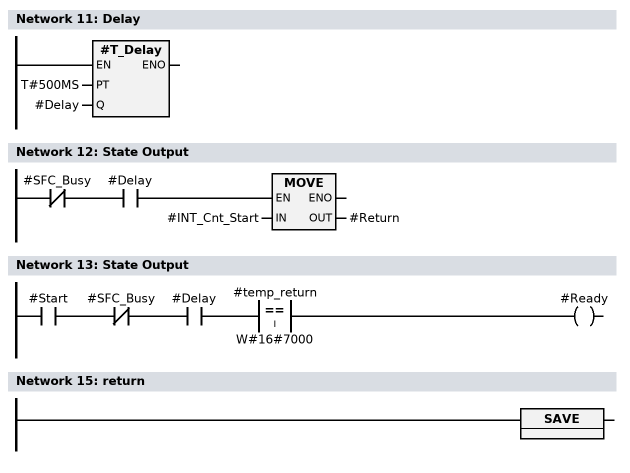
[picture p165: READ_DBL networks 11-15]
NETWORK
TITLE = Delay
      CALL  #T_Delay (
           PT                       := T#500MS,
           Q                        := #Delay);
      NOP   0;
NETWORK
TITLE = State Output
      AN    #SFC_Busy;
      A     #Delay;
      JNB   _007;
      L     #INT_Cnt_Start;
      T     #Return;
_007: NOP   0;
NETWORK
TITLE = State Output
      A     #Start;
      AN    #SFC_Busy;
      A     #Delay;
      A(;
      L     #temp_return;
      L     W#16#7000;
      ==I;
      );
      =     #Ready;
NETWORK
TITLE = restore register
      OPN   DB [#SysSave.DBNO];
      OPN   DI [#SysSave.DINO];
      LAR1  #SysSave.AR1;
      LAR2  #SysSave.AR2;
NETWORK
TITLE = return
      SET;
      SAVE;
END_FUNCTION_BLOCK

FUNCTION_BLOCK "WRITE_DBL"	// FB 193
TITLE = write to db on memory-card
//source-DB is on workarea of memory
//target-DB is on memory-card
VERSION : 0.1
VAR_INPUT
  DB_source : INT ;
  DB_target : INT ;
  Length : INT ;
  Start : BOOL ;
END_VAR
VAR_OUTPUT
  Return : INT ;
  Ready : BOOL ;
END_VAR
VAR
  imp_start : BOOL ;
  busy : BOOL ;
  puls_plus : BOOL ;
  puls_minus : BOOL ;
END_VAR
VAR_TEMP
  any_source : ANY ;
  any_target : ANY ;
  temp_rturn : INT ;
END_VAR
BEGIN
NETWORK
TITLE = create anypointer to source and target
//any to source
      L     W#16#1002;	//anytyp byte
      T     LW 0;
      L     #Length;	//number of bytes
      T     LW 2;
      L     #DB_source;	//number of DB-source 
      T     LW 4;
      L     0;	//begin in DB-source = byte 0
      SLD   3;
      OD    DW#16#84000000;	//constant
      T     LD 6;
//any to target
      L     W#16#1002;	//anytyp byte
      T     LW 10;
      L     #Length;	//number of bytes
      T     LW 12;
      L     #DB_target;	//number of DB-target
      T     LW 14;
      L     0;	//begin in DB-source = byte 0
      SLD   3;
      OD    DW#16#84000000;	//constant
      T     LD 16;
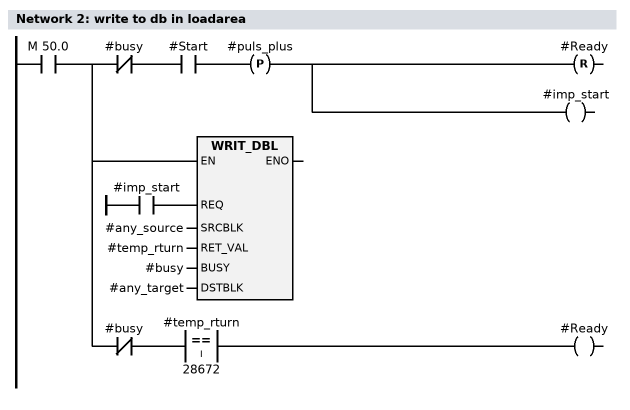
NETWORK
TITLE = write to db in loadarea
      A     M 50.0;
      =     L 22.0;
      A     L 22.0;
      AN    #busy;
      A(;
      A     #Start;
      BLD   100;
      FP    #puls_plus;
      );
      R     #Ready;
      =     #imp_start;
      A     #imp_start;
      =     L 22.1;
      BLD   103;
      A     L 22.0;
      JNB   _001;
      CALL  "WRIT_DBL" (
           REQ                      := L 22.1,
           SRCBLK                   := #any_source,
           RET_VAL                  := #temp_rturn,
           BUSY                     := #busy,
           DSTBLK                   := #any_target);
_001: NOP   0;
      A     L 22.0;
      AN    #busy;
      A(;
      L     #temp_rturn;
      L     28672;
      ==I;
      );
      =     #Ready;
END_FUNCTION_BLOCK

// FB 215: know-how protected block, not included

// FB 219: know-how protected block, not included

// FB 225: know-how protected block, not included

// FB 226: know-how protected block, not included

// FB 272: know-how protected block, not included

// FB 273: know-how protected block, not included

// FB 274: know-how protected block, not included

// FB 275: know-how protected block, not included

// FB 276: know-how protected block, not included

// FB 277: know-how protected block, not included

// FB 278: know-how protected block, not included

// FB 279: know-how protected block, not included

// FB 280: know-how protected block, not included

// FB 281: know-how protected block, not included

// FB 282: know-how protected block, not included

// FB 283: know-how protected block, not included

// FB 284: know-how protected block, not included

// FB 285: know-how protected block, not included

// FB 286: know-how protected block, not included

// FB 287: know-how protected block, not included

// FC 1: know-how protected block, not included

FUNCTION "Init" : VOID	// FC 2
TITLE = Program/PLC Init
VERSION : 0.1
VAR_TEMP
  ON : BOOL ;
  OFF : BOOL ;
END_VAR
BEGIN
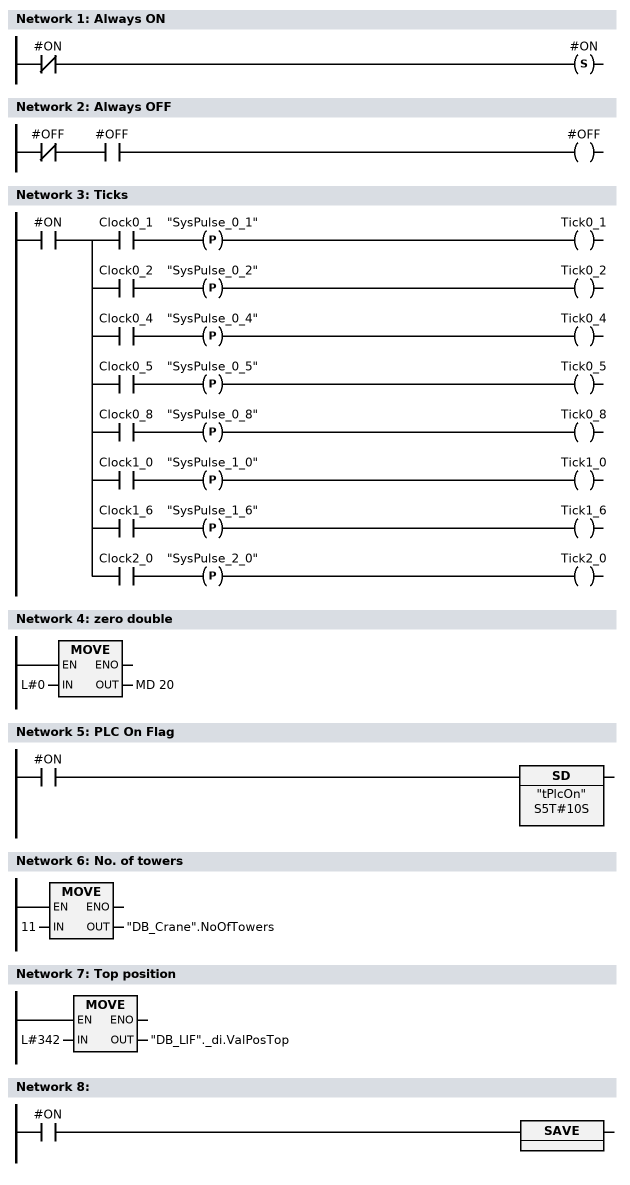
NETWORK
TITLE = Always ON
      AN    #ON;
      S     #ON;
NETWORK
TITLE = Always OFF
      AN    #OFF;
      A     #OFF;
      =     #OFF;
NETWORK
TITLE = Ticks
      A     #ON;
      =     L 1.0;
      A     L 1.0;
      A     "Clock0_1";
      FP    "SysPulse_0_1";
      =     "Tick0_1";
      A     L 1.0;
      A     "Clock0_2";
      FP    "SysPulse_0_2";
      =     "Tick0_2";
      A     L 1.0;
      A     "Clock0_4";
      FP    "SysPulse_0_4";
      =     "Tick0_4";
      A     L 1.0;
      A     "Clock0_5";
      FP    "SysPulse_0_5";
      =     "Tick0_5";
      A     L 1.0;
      A     "Clock0_8";
      FP    "SysPulse_0_8";
      =     "Tick0_8";
      A     L 1.0;
      A     "Clock1_0";
      FP    "SysPulse_1_0";
      =     "Tick1_0";
      A     L 1.0;
      A     "Clock1_6";
      FP    "SysPulse_1_6";
      =     "Tick1_6";
      A     L 1.0;
      A     "Clock2_0";
      FP    "SysPulse_2_0";
      =     "Tick2_0";
NETWORK
TITLE = zero double
      L     L#0;
      T     MD 20;
      NOP   0;
NETWORK
TITLE = PLC On Flag
      A     #ON;
      L     S5T#10S;
      SD    "tPlcOn";
NETWORK
TITLE = No. of towers
      L     11;
      T     "DB_Crane".NoOfTowers;
      NOP   0;
NETWORK
TITLE = Top position
      L     L#342;
      T     "DB_LIF"._di.ValPosTop;
      NOP   0;
NETWORK
TITLE =
      A     #ON;
      SAVE;
END_FUNCTION

// FC 5: know-how protected block, not included

// FC 6: know-how protected block, not included

// FC 8: know-how protected block, not included

FUNCTION "OpHours" : VOID	// FC 9
VERSION : 0.1
VAR_INPUT
  IN_xMoving : BOOL ;
  IN_xTick_1sec : BOOL ;
  IN_xResetServHours : BOOL ;
  IN_diServHoursPrest : DINT ;
END_VAR
VAR_IN_OUT
  INOUT_iWorkSec : INT ;
  INOUT_iServSec : INT ;
  INOUT_diWorkHours : DINT ;
  INOUT_diServHours : DINT ;
END_VAR
BEGIN
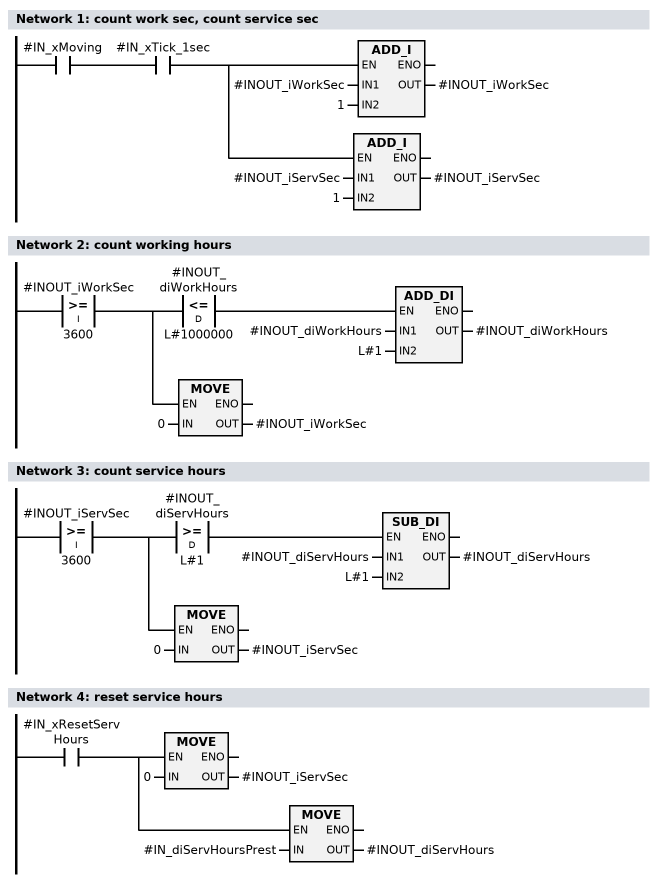
NETWORK
TITLE = count work sec, count service sec
      A     #IN_xMoving;
      A     #IN_xTick_1sec;
      =     L 0.0;
      A     L 0.0;
      JNB   _001;
      L     #INOUT_iWorkSec;
      L     1;
      +I;
      T     #INOUT_iWorkSec;
_001: NOP   0;
      A     L 0.0;
      JNB   _002;
      L     #INOUT_iServSec;
      L     1;
      +I;
      T     #INOUT_iServSec;
_002: NOP   0;
NETWORK
TITLE = count working hours
      L     #INOUT_iWorkSec;
      L     3600;
      >=I;
      =     L 0.0;
      A     L 0.0;
      A(;
      L     #INOUT_diWorkHours;
      L     L#1000000;
      <=D;
      );
      JNB   _003;
      L     #INOUT_diWorkHours;
      L     L#1;
      +D;
      T     #INOUT_diWorkHours;
_003: NOP   0;
      A     L 0.0;
      JNB   _004;
      L     0;
      T     #INOUT_iWorkSec;
_004: NOP   0;
NETWORK
TITLE = count service hours
      L     #INOUT_iServSec;
      L     3600;
      >=I;
      =     L 0.0;
      A     L 0.0;
      A(;
      L     #INOUT_diServHours;
      L     L#1;
      >=D;
      );
      JNB   _005;
      L     #INOUT_diServHours;
      L     L#1;
      -D;
      T     #INOUT_diServHours;
_005: NOP   0;
      A     L 0.0;
      JNB   _006;
      L     0;
      T     #INOUT_iServSec;
_006: NOP   0;
NETWORK
TITLE = reset service hours
      A     #IN_xResetServHours;
      =     L 0.0;
      A     L 0.0;
      JNB   _007;
      L     0;
      T     #INOUT_iServSec;
_007: NOP   0;
      A     L 0.0;
      JNB   _008;
      L     #IN_diServHoursPrest;
      T     #INOUT_diServHours;
_008: NOP   0;
END_FUNCTION

// FC 10: know-how protected block, not included

FUNCTION "AbsEncoder" : VOID	// FC 11
TITLE = AbsEncoder
//calculate position value depend from encoder resolution
VERSION : 0.1
VAR_INPUT
  IN_DW_ProcessData : DWORD ;
  IN_DINT_Turn100 : DINT ;
  IN_DINT_PresetVal : DINT ;
  IN_Resolution_4096 : BOOL ;
  IN_Resolution_8192 : BOOL ;
  IN_BOOL_Preset : BOOL ;
END_VAR
VAR_OUTPUT
  OUT_DINT_EncMm : DINT ;
  OUT_DW_ProcessData : DWORD ;
END_VAR
VAR_TEMP
  TEMP_DINT_WayByFullTurns : DINT ;
  TEMP_DINT_WayByActTurn : DINT ;
  TEMP_DINT_Resolution : DINT ;
  TEMP_DW_01 : DWORD ;
  TEMP_DW_00 : DWORD ;
  TEMP_DW_Mask1 : DWORD ;
  TEMP_W_Mask2 : WORD ;
  TEMP_DW_Mask3 : DWORD ;
  TEMP_DINT_00 : DINT ;
  TEMP_DINT_PresetTurns : DINT ;
  TEMP_DINT_PresetVal100 : DINT ;
  TEMP_DINT_PresetAngle : DINT ;
  ON : BOOL ;
  TEMP_BOOL_RetValFault : BOOL ;
END_VAR
BEGIN
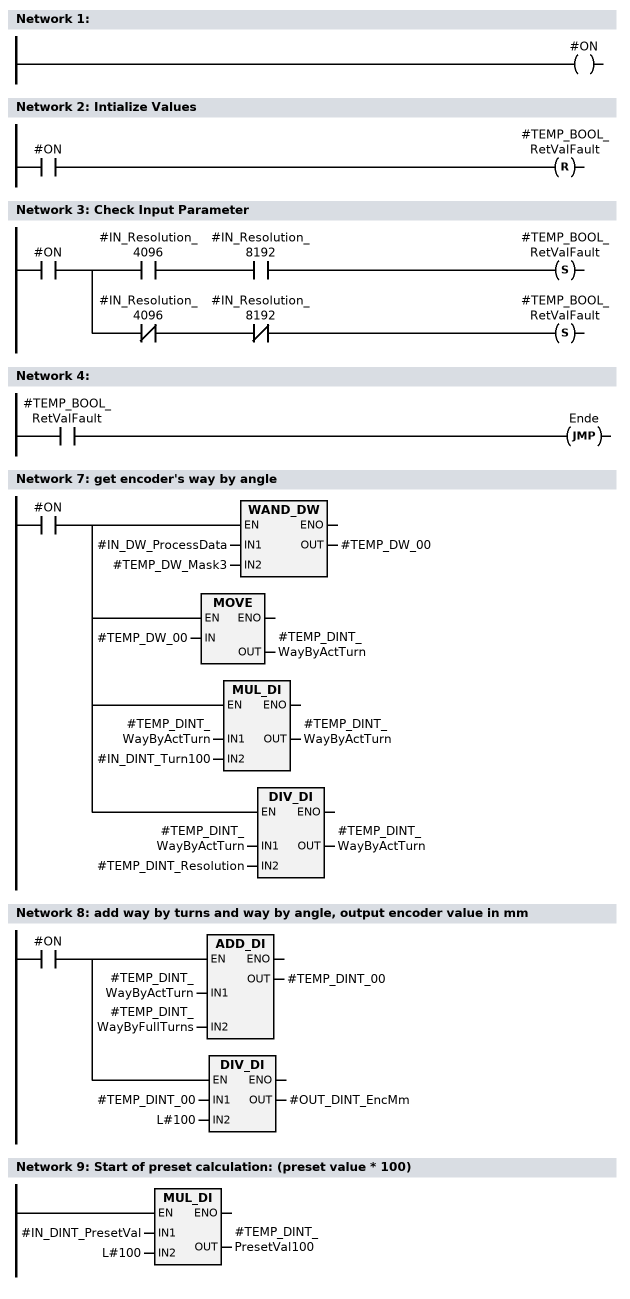
NETWORK
TITLE =
      SET;
      =     #ON;
NETWORK
TITLE = Intialize Values
      A     #ON;
      R     #TEMP_BOOL_RetValFault;
NETWORK
TITLE = Check Input Parameter
      A     #ON;
      =     L 47.0;
      A     L 47.0;
      A     #IN_Resolution_4096;
      A     #IN_Resolution_8192;
      S     #TEMP_BOOL_RetValFault;
      A     L 47.0;
      AN    #IN_Resolution_4096;
      AN    #IN_Resolution_8192;
      S     #TEMP_BOOL_RetValFault;
NETWORK
TITLE =
      A     #TEMP_BOOL_RetValFault;
      JC    Ende;
NETWORK
TITLE =
      A     #ON;
      =     L 47.0;
      A     L 47.0;
      A     #IN_Resolution_4096;
      =     L 47.1;
      A(;
      A(;
      A     L 47.1;
      JNB   _001;
      L     DW#16#1FFF000;
      T     #TEMP_DW_Mask1;
      SET;
      SAVE;
      CLR;
_001: A     BR;
      );
      JNB   _002;
      L     W#16#C;
      T     #TEMP_W_Mask2;
      SET;
      SAVE;
      CLR;
_002: A     BR;
      );
      JNB   _003;
      L     DW#16#FFF;
      T     #TEMP_DW_Mask3;
_003: NOP   0;
      A     L 47.1;
      JNB   _004;
      L     L#4096;
      T     #TEMP_DINT_Resolution;
_004: NOP   0;
      A     L 47.0;
      A     #IN_Resolution_8192;
      =     L 47.1;
      A(;
      A(;
      A     L 47.1;
      JNB   _005;
      L     DW#16#1FFE000;
      T     #TEMP_DW_Mask1;
      SET;
      SAVE;
      CLR;
_005: A     BR;
      );
      JNB   _006;
      L     W#16#D;
      T     #TEMP_W_Mask2;
      SET;
      SAVE;
      CLR;
_006: A     BR;
      );
      JNB   _007;
      L     DW#16#1FFF;
      T     #TEMP_DW_Mask3;
_007: NOP   0;
      A     L 47.1;
      JNB   _008;
      L     L#8192;
      T     #TEMP_DINT_Resolution;
_008: NOP   0;
NETWORK
TITLE = Start of actual mm-calculation: get encoder's way by full turns
      A     #ON;
      =     L 47.0;
      A     L 47.0;
      JNB   _009;
      L     #IN_DW_ProcessData;
      L     #TEMP_DW_Mask1;
      AD;
      T     #TEMP_DW_00;
_009: NOP   0;
      A     L 47.0;
      JNB   _00a;
      L     #TEMP_W_Mask2;
      L     #TEMP_DW_00;
      SRD;
      T     #TEMP_DW_00;
_00a: NOP   0;
      A     L 47.0;
      JNB   _00b;
      L     #TEMP_DW_00;
      T     #TEMP_DINT_WayByFullTurns;
_00b: NOP   0;
      A     L 47.0;
      JNB   _00c;
      L     #TEMP_DINT_WayByFullTurns;
      L     #IN_DINT_Turn100;
      *D;
      T     #TEMP_DINT_WayByFullTurns;
_00c: NOP   0;
NETWORK
TITLE = get encoder's way by angle
      A     #ON;
      =     L 47.0;
      A     L 47.0;
      JNB   _00d;
      L     #IN_DW_ProcessData;
      L     #TEMP_DW_Mask3;
      AD;
      T     #TEMP_DW_00;
_00d: NOP   0;
      A     L 47.0;
      JNB   _00e;
      L     #TEMP_DW_00;
      T     #TEMP_DINT_WayByActTurn;
_00e: NOP   0;
      A     L 47.0;
      JNB   _00f;
      L     #TEMP_DINT_WayByActTurn;
      L     #IN_DINT_Turn100;
      *D;
      T     #TEMP_DINT_WayByActTurn;
_00f: NOP   0;
      A     L 47.0;
      JNB   _010;
      L     #TEMP_DINT_WayByActTurn;
      L     #TEMP_DINT_Resolution;
      /D;
      T     #TEMP_DINT_WayByActTurn;
_010: NOP   0;
NETWORK
TITLE = add way by turns and way by angle, output encoder value in mm
      A     #ON;
      =     L 47.0;
      A     L 47.0;
      JNB   _011;
      L     #TEMP_DINT_WayByActTurn;
      L     #TEMP_DINT_WayByFullTurns;
      +D;
      T     #TEMP_DINT_00;
_011: NOP   0;
      A     L 47.0;
      JNB   _012;
      L     #TEMP_DINT_00;
      L     L#100;
      /D;
      T     #OUT_DINT_EncMm;
_012: NOP   0;
NETWORK
TITLE = Start of preset calculation: (preset value * 100)
      L     #IN_DINT_PresetVal;
      L     L#100;
      *D;
      T     #TEMP_DINT_PresetVal100;
      NOP   0;
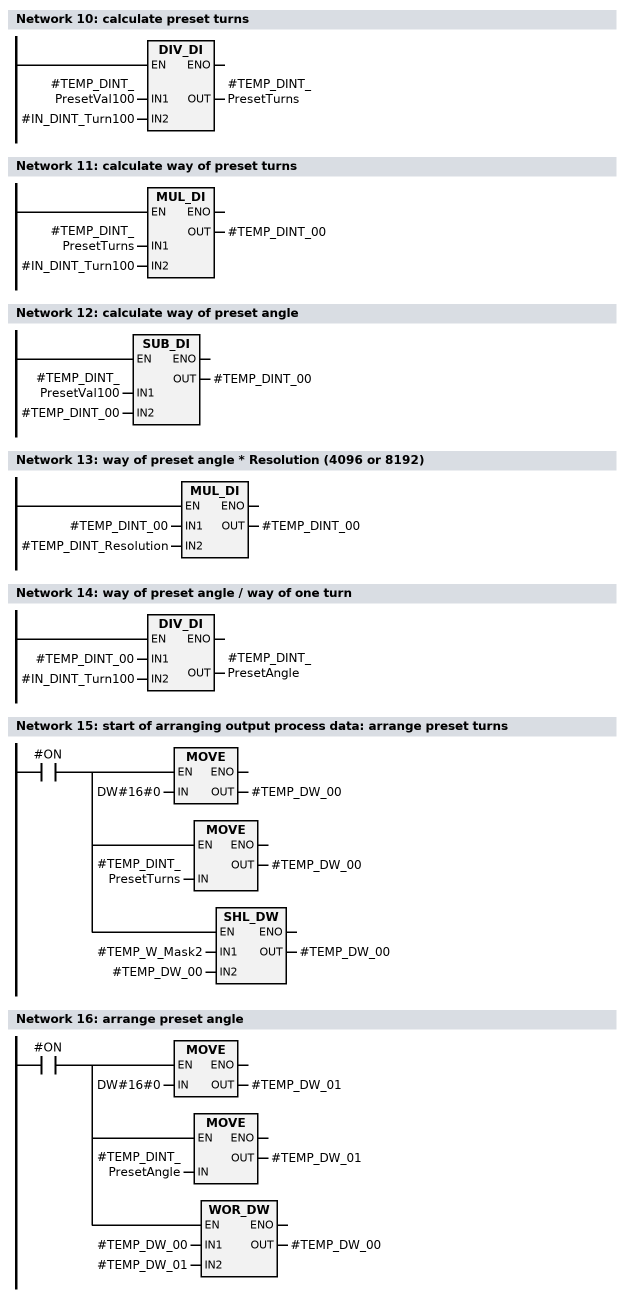
NETWORK
TITLE = calculate preset turns
      L     #TEMP_DINT_PresetVal100;
      L     #IN_DINT_Turn100;
      /D;
      T     #TEMP_DINT_PresetTurns;
      NOP   0;
NETWORK
TITLE = calculate way of preset turns
      L     #TEMP_DINT_PresetTurns;
      L     #IN_DINT_Turn100;
      *D;
      T     #TEMP_DINT_00;
      NOP   0;
NETWORK
TITLE = calculate way of preset angle 
      L     #TEMP_DINT_PresetVal100;
      L     #TEMP_DINT_00;
      -D;
      T     #TEMP_DINT_00;
      NOP   0;
NETWORK
TITLE = way of preset angle * Resolution (4096 or 8192)
      L     #TEMP_DINT_00;
      L     #TEMP_DINT_Resolution;
      *D;
      T     #TEMP_DINT_00;
      NOP   0;
NETWORK
TITLE = way of preset angle / way of one turn
      L     #TEMP_DINT_00;
      L     #IN_DINT_Turn100;
      /D;
      T     #TEMP_DINT_PresetAngle;
      NOP   0;
NETWORK
TITLE = start of arranging output process data: arrange preset turns
      A     #ON;
      =     L 47.0;
      A     L 47.0;
      JNB   _013;
      L     DW#16#0;
      T     #TEMP_DW_00;
_013: NOP   0;
      A     L 47.0;
      JNB   _014;
      L     #TEMP_DINT_PresetTurns;
      T     #TEMP_DW_00;
_014: NOP   0;
      A     L 47.0;
      JNB   _015;
      L     #TEMP_W_Mask2;
      L     #TEMP_DW_00;
      SLD;
      T     #TEMP_DW_00;
_015: NOP   0;
NETWORK
TITLE = arrange preset angle
      A     #ON;
      =     L 47.0;
      A     L 47.0;
      JNB   _016;
      L     DW#16#0;
      T     #TEMP_DW_01;
_016: NOP   0;
      A     L 47.0;
      JNB   _017;
      L     #TEMP_DINT_PresetAngle;
      T     #TEMP_DW_01;
_017: NOP   0;
      A     L 47.0;
      JNB   _018;
      L     #TEMP_DW_00;
      L     #TEMP_DW_01;
      OD;
      T     #TEMP_DW_00;
_018: NOP   0;
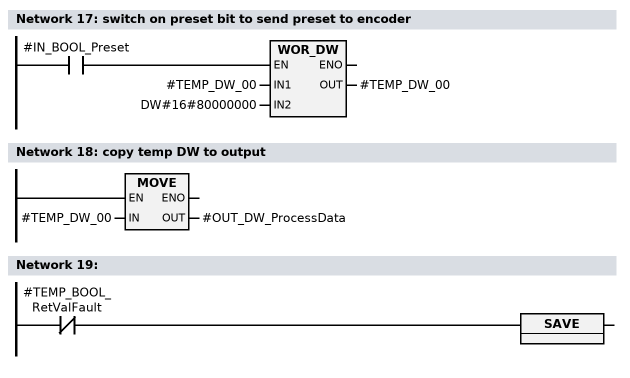
NETWORK
TITLE = switch on preset bit to send preset to encoder
      A     #IN_BOOL_Preset;
      JNB   _019;
      L     #TEMP_DW_00;
      L     DW#16#80000000;
      OD;
      T     #TEMP_DW_00;
_019: NOP   0;
NETWORK
TITLE = copy temp DW to output 
      L     #TEMP_DW_00;
      T     #OUT_DW_ProcessData;
      NOP   0;
NETWORK
TITLE =
Ende: AN    #TEMP_BOOL_RetValFault;
      SAVE;
END_FUNCTION

FUNCTION "Motor_2_frequ" : VOID	// FC 12
VERSION : 0.1
VAR_INPUT
  IN_x_Release : BOOL ;
  IN_BOOL_ServLeft : BOOL ;
  IN_BOOL_ServRight : BOOL ;
  IN_BOOL_ServMode : BOOL ;
  IN_StartPosMode : BOOL ;
  IN_TargetVal : DINT ;
  IN_ActPos : DINT ;
  IN_SlowWin : DINT ;
  IN_StopWin : DINT ;
  IN_PosWin : DINT ;
END_VAR
VAR_OUTPUT
  OUT_BOOL_FastFrequ : BOOL ;
  OUT_BOOL_Pos_OK : BOOL ;
END_VAR
VAR_IN_OUT
  INOUT_x_Minus : BOOL ;
  INOUT_x_Plus : BOOL ;
END_VAR
VAR_TEMP
  TEMP_DINT_00 : DINT ;
  TMP_x_InPosition : BOOL ;
  TMP_x_Slow : BOOL ;
  TMP_x_PosOk : BOOL ;
END_VAR
BEGIN
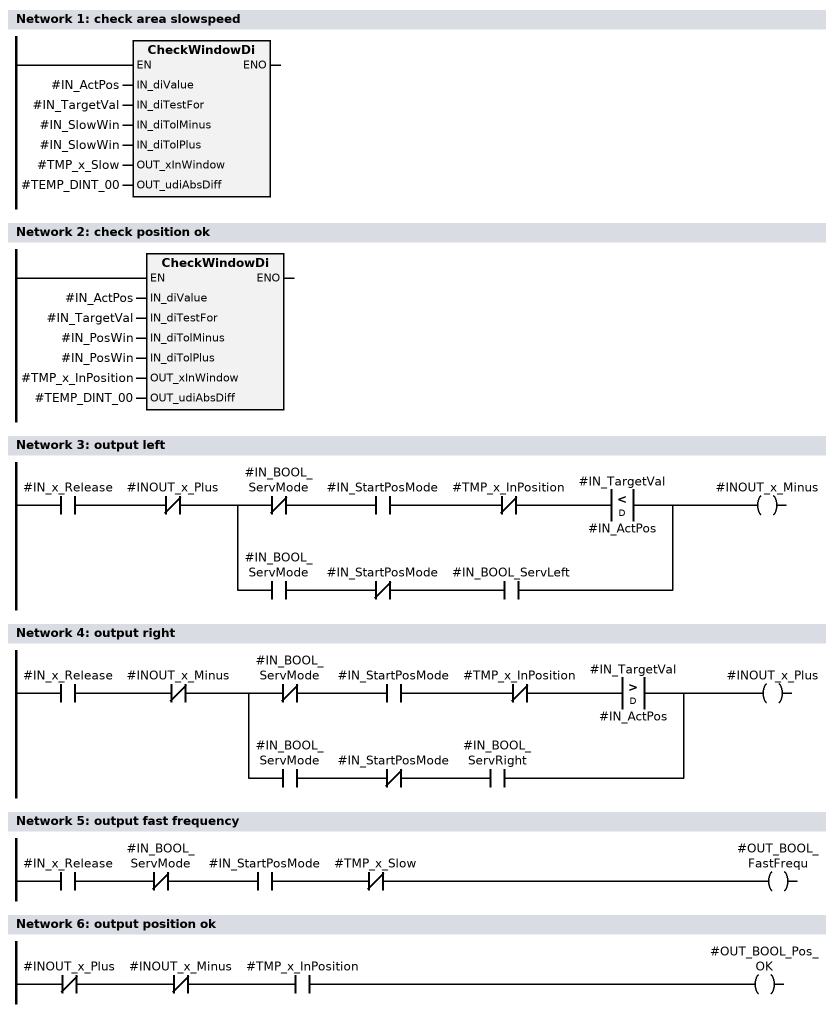
NETWORK
TITLE = check area slowspeed
      CALL  "CheckWindowDi" (
           IN_diValue               := #IN_ActPos,
           IN_diTestFor             := #IN_TargetVal,
           IN_diTolMinus            := #IN_SlowWin,
           IN_diTolPlus             := #IN_SlowWin,
           OUT_xInWindow            := #TMP_x_Slow,
           OUT_udiAbsDiff           := #TEMP_DINT_00);
      NOP   0;
NETWORK
TITLE = check position ok
      CALL  "CheckWindowDi" (
           IN_diValue               := #IN_ActPos,
           IN_diTestFor             := #IN_TargetVal,
           IN_diTolMinus            := #IN_PosWin,
           IN_diTolPlus             := #IN_PosWin,
           OUT_xInWindow            := #TMP_x_InPosition,
           OUT_udiAbsDiff           := #TEMP_DINT_00);
      NOP   0;
NETWORK
TITLE = output left
      A     #IN_x_Release;
      AN    #INOUT_x_Plus;
      A(;
      AN    #IN_BOOL_ServMode;
      A     #IN_StartPosMode;
      AN    #TMP_x_InPosition;
      A(;
      L     #IN_TargetVal;
      L     #IN_ActPos;
      <D;
      );
      O;
      A     #IN_BOOL_ServMode;
      AN    #IN_StartPosMode;
      A     #IN_BOOL_ServLeft;
      );
      =     #INOUT_x_Minus;
NETWORK
TITLE = output right
      A     #IN_x_Release;
      AN    #INOUT_x_Minus;
      A(;
      AN    #IN_BOOL_ServMode;
      A     #IN_StartPosMode;
      AN    #TMP_x_InPosition;
      A(;
      L     #IN_TargetVal;
      L     #IN_ActPos;
      >D;
      );
      O;
      A     #IN_BOOL_ServMode;
      AN    #IN_StartPosMode;
      A     #IN_BOOL_ServRight;
      );
      =     #INOUT_x_Plus;
NETWORK
TITLE = output fast frequency 
      A     #IN_x_Release;
      AN    #IN_BOOL_ServMode;
      A     #IN_StartPosMode;
      AN    #TMP_x_Slow;
      =     #OUT_BOOL_FastFrequ;
NETWORK
TITLE = output position ok
      AN    #INOUT_x_Plus;
      AN    #INOUT_x_Minus;
      A     #TMP_x_InPosition;
      =     #OUT_BOOL_Pos_OK;
END_FUNCTION

// FC 15: know-how protected block, not included

FUNCTION "Scan_BRI" : VOID	// FC 21
TITLE = scan positions bridge
VERSION : 0.1
VAR_INPUT
  in_i_DBNo : INT ;
  in_i_ActRow : INT ;
  in_i_NoOfDataSets : INT ;
  in_di_DatSetLenght : DINT ;
  in_di_ActAxisPos : DINT ;
  in_di_DataStartByte : DINT ;
  in_di_AreaWin : DINT ;
  in_di_PosWin : DINT ;
END_VAR
VAR_OUTPUT
  out_i_SetNo : INT ;
  out_i_AreaNo : INT ;
  out_b_InArea : BOOL ;
  out_b_InPos : BOOL ;
  out_i_LIF_DBNo : INT ;
  out_i_LIF_DBNo_2 : INT ;
END_VAR
VAR_TEMP
  Save_AR1 : DWORD ;
  Save_AR2 : DWORD ;
  tmp_di_1 : DINT ;
  tmp_di_2 : DINT ;
  tmp_di_Pointer : DINT ;
  tmp_di_PosVal : DINT ;
  tmp_i_PosNo : INT ;
  tmp_i_PosNoVal : INT ;
  tmp_i_DBNo : INT ;
  tmp_i_1 : INT ;
  tmp_i_LIF_DBNo : INT ;
  tmp_i_LIF_DBNo_2 : INT ;
  tmp_i_offsetPointer : INT ;
  ON : BOOL ;
  OFF : BOOL ;
  tmp_b_LoopBrake : BOOL ;
  err_input : BOOL ;
END_VAR
BEGIN
NETWORK
TITLE = save register
      TAR1  #Save_AR1;
      TAR2  #Save_AR2;
NETWORK
TITLE = on/off
      SET;
      =     #ON;
      CLR;
      =     #OFF;
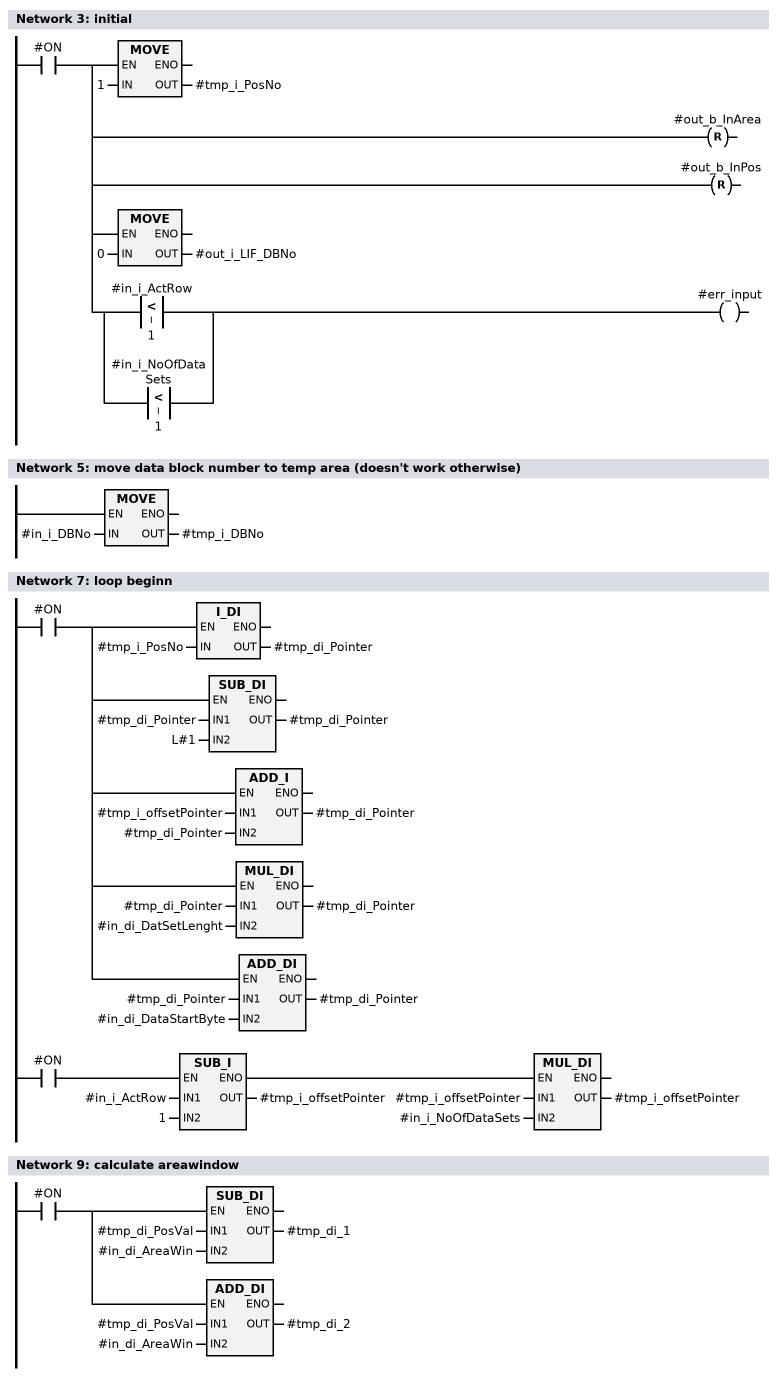
NETWORK
TITLE = initial
//set loopcounter to 0
//reset outputs
      A     #ON;
      =     L 40.0;
      A     L 40.0;
      JNB   _001;
      L     1;
      T     #tmp_i_PosNo;
_001: NOP   0;
      A     L 40.0;
      BLD   102;
      R     #out_b_InArea;
      A     L 40.0;
      BLD   102;
      R     #out_b_InPos;
      A     L 40.0;
      JNB   _002;
      L     0;
      T     #out_i_LIF_DBNo;
_002: NOP   0;
      A     L 40.0;
      A(;
      O(;
      L     #in_i_ActRow;
      L     1;
      <I;
      );
      O(;
      L     #in_i_NoOfDataSets;
      L     1;
      <I;
      );
      );
      =     #err_input;
NETWORK
TITLE =
      AN    #err_input;
      JC    NoEr;	// On Error CLR all Outputs
      L     0;
      T     #out_i_SetNo;
      T     #out_i_AreaNo;
      T     #out_i_LIF_DBNo;
      T     #out_i_LIF_DBNo_2;
      A     #OFF;
      =     #out_b_InArea;
      =     #out_b_InPos;
      BEU;
NoEr: NOP   0;
NETWORK
TITLE = move data block number to temp area (doesn't work otherwise)
//doesn't work otherwise
      L     #in_i_DBNo;
      T     #tmp_i_DBNo;
      NOP   0;
NETWORK
TITLE = open DB
      OPN   DB [#tmp_i_DBNo];
NETWORK
TITLE = loop beginn
//calculate pointer to positionvalue
//insert calculating rows [2016 TH]
scbr: A     #ON;
      =     L 39.0;
      A     L 39.0;
      JNB   _003;
      L     #tmp_i_PosNo;
      ITD;
      T     #tmp_di_Pointer;
_003: NOP   0;
      A     L 39.0;
      JNB   _004;
      L     #tmp_di_Pointer;
      L     L#1;
      -D;
      T     #tmp_di_Pointer;
_004: NOP   0;
      A(;
      A     L 39.0;
      JNB   _005;
      L     #in_i_ActRow;
      L     1;
      -I;
      T     #tmp_i_offsetPointer;
      AN    OV;
      SAVE;
      CLR;
_005: A     BR;
      );
      JNB   _006;
      L     #tmp_i_offsetPointer;
      L     #in_i_NoOfDataSets;
      *D;
      T     #tmp_i_offsetPointer;
_006: NOP   0;
      A     L 39.0;
      JNB   _007;
      L     #tmp_i_offsetPointer;
      L     #tmp_di_Pointer;
      +I;
      T     #tmp_di_Pointer;
_007: NOP   0;
      A     L 39.0;
      JNB   _008;
      L     #tmp_di_Pointer;
      L     #in_di_DatSetLenght;
      *D;
      T     #tmp_di_Pointer;
_008: NOP   0;
      A     L 39.0;
      JNB   _009;
      L     #tmp_di_Pointer;
      L     #in_di_DataStartByte;
      +D;
      T     #tmp_di_Pointer;
_009: NOP   0;
NETWORK
TITLE = get positionvalue 
      L     #tmp_di_Pointer;	// load pointer
      SLD   3;	// shift left 3 bits to achieve pointer format
      LAR1;	// load adressregister 1 with pointer
      L     DBD [AR1,P#2.0];	// load position from DataBlock
      T     #tmp_di_PosVal;	// Transfer to temp for window check
      L     DBW [AR1,P#0.0];
      T     #tmp_i_PosNoVal;
      L     DBW [AR1,P#6.0];	// LIF DB number
      T     #tmp_i_LIF_DBNo;
      L     DBW [AR1,P#8.0];	// LIF DB number
      T     #tmp_i_LIF_DBNo_2;
NETWORK
TITLE = calculate areawindow
      A     #ON;
      =     L 40.0;
      A     L 40.0;
      JNB   _00a;
      L     #tmp_di_PosVal;
      L     #in_di_AreaWin;
      -D;
      T     #tmp_di_1;
_00a: NOP   0;
      A     L 40.0;
      JNB   _00b;
      L     #tmp_di_PosVal;
      L     #in_di_AreaWin;
      +D;
      T     #tmp_di_2;
_00b: NOP   0;
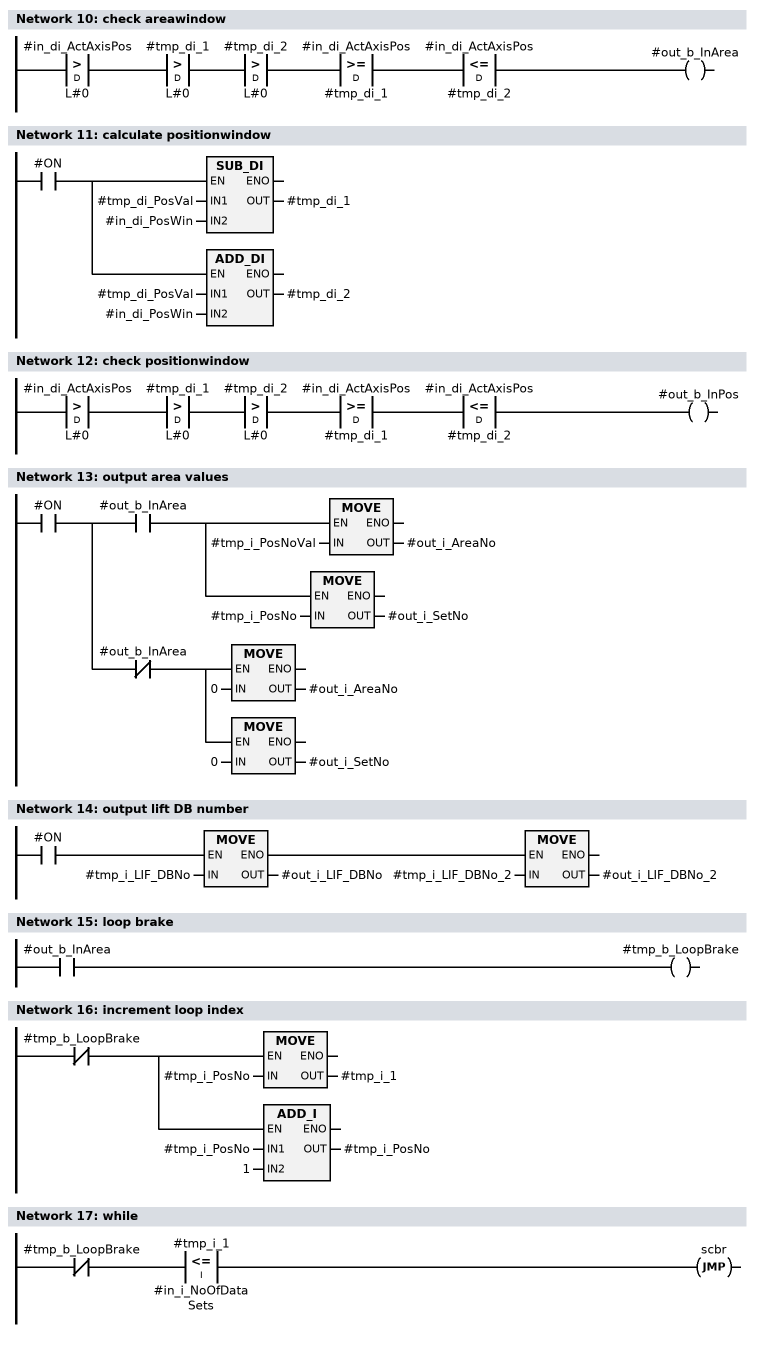
NETWORK
TITLE = check areawindow
      A(;
      L     #in_di_ActAxisPos;
      L     L#0;
      >D;
      );
      A(;
      L     #tmp_di_1;
      L     L#0;
      >D;
      );
      A(;
      L     #tmp_di_2;
      L     L#0;
      >D;
      );
      A(;
      L     #in_di_ActAxisPos;
      L     #tmp_di_1;
      >=D;
      );
      A(;
      L     #in_di_ActAxisPos;
      L     #tmp_di_2;
      <=D;
      );
      =     #out_b_InArea;
NETWORK
TITLE = calculate positionwindow
      A     #ON;
      =     L 40.0;
      A     L 40.0;
      JNB   _00c;
      L     #tmp_di_PosVal;
      L     #in_di_PosWin;
      -D;
      T     #tmp_di_1;
_00c: NOP   0;
      A     L 40.0;
      JNB   _00d;
      L     #tmp_di_PosVal;
      L     #in_di_PosWin;
      +D;
      T     #tmp_di_2;
_00d: NOP   0;
NETWORK
TITLE = check positionwindow
      A(;
      L     #in_di_ActAxisPos;
      L     L#0;
      >D;
      );
      A(;
      L     #tmp_di_1;
      L     L#0;
      >D;
      );
      A(;
      L     #tmp_di_2;
      L     L#0;
      >D;
      );
      A(;
      L     #in_di_ActAxisPos;
      L     #tmp_di_1;
      >=D;
      );
      A(;
      L     #in_di_ActAxisPos;
      L     #tmp_di_2;
      <=D;
      );
      =     #out_b_InPos;
NETWORK
TITLE = output area values
      A     #ON;
      =     L 40.0;
      A     L 40.0;
      A     #out_b_InArea;
      =     L 40.1;
      A     L 40.1;
      JNB   _00e;
      L     #tmp_i_PosNoVal;
      T     #out_i_AreaNo;
_00e: NOP   0;
      A     L 40.1;
      JNB   _00f;
      L     #tmp_i_PosNo;
      T     #out_i_SetNo;
_00f: NOP   0;
      A     L 40.0;
      AN    #out_b_InArea;
      =     L 40.1;
      A     L 40.1;
      JNB   _010;
      L     0;
      T     #out_i_AreaNo;
_010: NOP   0;
      A     L 40.1;
      JNB   _011;
      L     0;
      T     #out_i_SetNo;
_011: NOP   0;
NETWORK
TITLE = output lift DB number
      A(;
      A     #ON;
      JNB   _012;
      L     #tmp_i_LIF_DBNo;
      T     #out_i_LIF_DBNo;
      SET;
      SAVE;
      CLR;
_012: A     BR;
      );
      JNB   _013;
      L     #tmp_i_LIF_DBNo_2;
      T     #out_i_LIF_DBNo_2;
_013: NOP   0;
NETWORK
TITLE = loop brake
      A     #out_b_InArea;
      =     #tmp_b_LoopBrake;
NETWORK
TITLE = increment loop index
      AN    #tmp_b_LoopBrake;
      =     L 40.0;
      A     L 40.0;
      JNB   _014;
      L     #tmp_i_PosNo;
      T     #tmp_i_1;
_014: NOP   0;
      A     L 40.0;
      JNB   _015;
      L     #tmp_i_PosNo;
      L     1;
      +I;
      T     #tmp_i_PosNo;
_015: NOP   0;
NETWORK
TITLE = while 
      AN    #tmp_b_LoopBrake;
      A(;
      L     #tmp_i_1;
      L     #in_i_NoOfDataSets;
      <=I;
      );
      JC    scbr;
NETWORK
TITLE = restore register
      LAR1  #Save_AR1;
      LAR2  #Save_AR2;
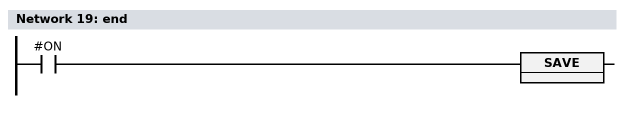
NETWORK
TITLE = end
      A     #ON;
      SAVE;
END_FUNCTION

FUNCTION "Scan_BRI_MAN" : VOID	// FC 22
TITLE = scan positions bridge
VERSION : 1.0
VAR_INPUT
  in_i_DBNo : INT ;
  in_i_ActRow : INT ;
  in_i_NoOfDataSets : INT ;
  in_di_DatSetLenght : DINT ;
  in_di_DataStartByte : DINT ;
  in_di_ActAxisPos : DINT ;
END_VAR
VAR_OUTPUT
  out_di_PrevPos : DINT ;
  out_di_ActPos : DINT ;
  out_di_NextPos : DINT ;
  out_di_MinPos : DINT ;
  out_di_MaxPos : DINT ;
  out_i_PrevPosNo : INT ;
  out_i_NextPosNo : INT ;
  out_i_MinPosNo : INT ;
  out_i_MaxPosNo : INT ;
END_VAR
VAR_TEMP
  Save_AR1 : DWORD ;
  Save_AR2 : DWORD ;
  tmp_di_1 : DINT ;
  tmp_di_Pointer : DINT ;
  tmp_di_PosVal : DINT ;
  tmp_di_PosData : DINT ;
  tmp_di_PosDataPlus : DINT ;
  tmp_di_PosDataMinus : DINT ;
  tmp_di_PosDataLow : DINT ;
  tmp_di_PosDataHigh : DINT ;
  tmp_di_PrevPos : DINT ;
  tmp_di_NextPos : DINT ;
  tmp_i_Counter : INT ;
  tmp_i_DBNo : INT ;
  tmp_i_PosNo : INT ;
  tmp_i_PosDataNo : INT ;
  tmp_i_PrevPosNo : INT ;
  tmp_i_NextPosNo : INT ;
  tmp_i_MinPosNo : INT ;
  tmp_i_MaxPosNo : INT ;
  tmp_i_1 : INT ;
  tmp_i_offsetPointer : INT ;
  TEMP1 : BOOL ;
  ON : BOOL ;
  OFF : BOOL ;
  err_input : BOOL ;
END_VAR
BEGIN
NETWORK
TITLE = save register
      TAR1  #Save_AR1;
      TAR2  #Save_AR2;
NETWORK
TITLE = on/off
      SET;
      =     #ON;
      CLR;
      =     #OFF;
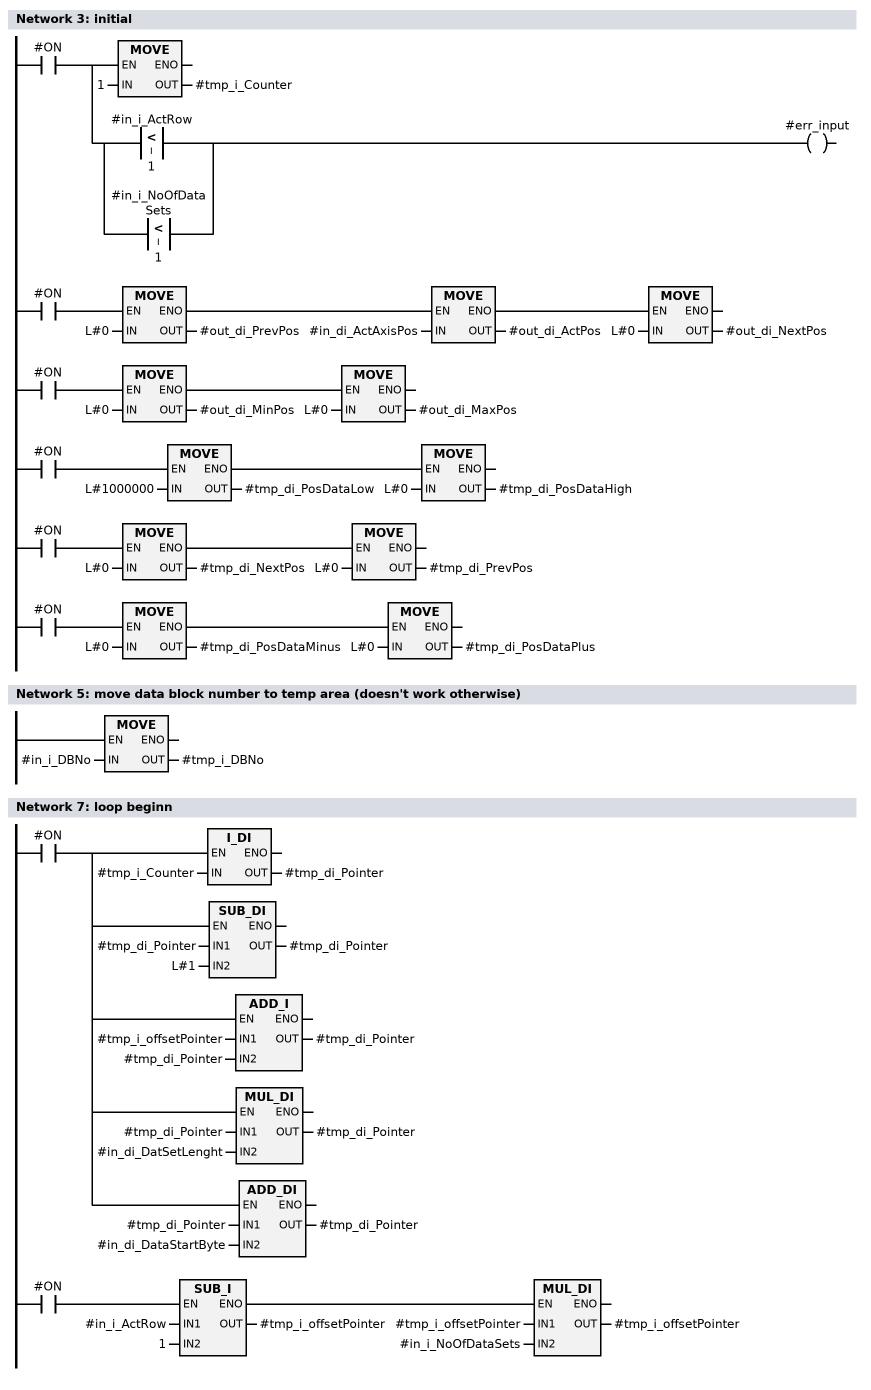
NETWORK
TITLE = initial
//set loopcounter to 0
//reset outputs
      A     #ON;
      =     L 70.0;
      A     L 70.0;
      JNB   _001;
      L     1;
      T     #tmp_i_Counter;
_001: NOP   0;
      A(;
      A(;
      A     L 70.0;
      JNB   _002;
      L     L#0;
      T     #out_di_PrevPos;
      SET;
      SAVE;
      CLR;
_002: A     BR;
      );
      JNB   _003;
      L     #in_di_ActAxisPos;
      T     #out_di_ActPos;
      SET;
      SAVE;
      CLR;
_003: A     BR;
      );
      JNB   _004;
      L     L#0;
      T     #out_di_NextPos;
_004: NOP   0;
      A(;
      A     L 70.0;
      JNB   _005;
      L     L#0;
      T     #out_di_MinPos;
      SET;
      SAVE;
      CLR;
_005: A     BR;
      );
      JNB   _006;
      L     L#0;
      T     #out_di_MaxPos;
_006: NOP   0;
      A(;
      A     L 70.0;
      JNB   _007;
      L     L#1000000;
      T     #tmp_di_PosDataLow;
      SET;
      SAVE;
      CLR;
_007: A     BR;
      );
      JNB   _008;
      L     L#0;
      T     #tmp_di_PosDataHigh;
_008: NOP   0;
      A(;
      A     L 70.0;
      JNB   _009;
      L     L#0;
      T     #tmp_di_NextPos;
      SET;
      SAVE;
      CLR;
_009: A     BR;
      );
      JNB   _00a;
      L     L#0;
      T     #tmp_di_PrevPos;
_00a: NOP   0;
      A(;
      A     L 70.0;
      JNB   _00b;
      L     L#0;
      T     #tmp_di_PosDataMinus;
      SET;
      SAVE;
      CLR;
_00b: A     BR;
      );
      JNB   _00c;
      L     L#0;
      T     #tmp_di_PosDataPlus;
_00c: NOP   0;
      A     L 70.0;
      A(;
      O(;
      L     #in_i_ActRow;
      L     1;
      <I;
      );
      O(;
      L     #in_i_NoOfDataSets;
      L     1;
      <I;
      );
      );
      =     #err_input;
NETWORK
TITLE =
      AN    #err_input;
      JC    NoEr;	// On Error CLR all Outputs
      BEU;
NoEr: NOP   0;
NETWORK
TITLE = move data block number to temp area (doesn't work otherwise)
//doesn't work otherwise
      L     #in_i_DBNo;
      T     #tmp_i_DBNo;
      NOP   0;
NETWORK
TITLE = open DB
      OPN   DB [#tmp_i_DBNo];
NETWORK
TITLE = loop beginn
//calculate pointer to positionvalue
scbr: A     #ON;
      =     L 69.0;
      A     L 69.0;
      JNB   _00d;
      L     #tmp_i_Counter;
      ITD;
      T     #tmp_di_Pointer;
_00d: NOP   0;
      A     L 69.0;
      JNB   _00e;
      L     #tmp_di_Pointer;
      L     L#1;
      -D;
      T     #tmp_di_Pointer;
_00e: NOP   0;
      A(;
      A     L 69.0;
      JNB   _00f;
      L     #in_i_ActRow;
      L     1;
      -I;
      T     #tmp_i_offsetPointer;
      AN    OV;
      SAVE;
      CLR;
_00f: A     BR;
      );
      JNB   _010;
      L     #tmp_i_offsetPointer;
      L     #in_i_NoOfDataSets;
      *D;
      T     #tmp_i_offsetPointer;
_010: NOP   0;
      A     L 69.0;
      JNB   _027;
      L     #tmp_i_offsetPointer;
      L     #tmp_di_Pointer;
      +I;
      T     #tmp_di_Pointer;
_027: NOP   0;
      A     L 69.0;
      JNB   _028;
      L     #tmp_di_Pointer;
      L     #in_di_DatSetLenght;
      *D;
      T     #tmp_di_Pointer;
_028: NOP   0;
      A     L 69.0;
      JNB   _029;
      L     #tmp_di_Pointer;
      L     #in_di_DataStartByte;
      +D;
      T     #tmp_di_Pointer;
_029: NOP   0;
NETWORK
TITLE = get positionvalue 
      L     #tmp_di_Pointer;	// load pointer
      SLD   3;	// shift left 3 bits to achieve pointer format
      LAR1;	// load adressregister 1 with pointer
      L     DBD [AR1,P#2.0];	// load position from DataBlock
      T     #tmp_di_PosVal;	// Transfer to temp for window check
      L     DBW [AR1,P#0.0];	// load position number from DataBlock
      T     #tmp_i_PosNo;	// Transfer to temp
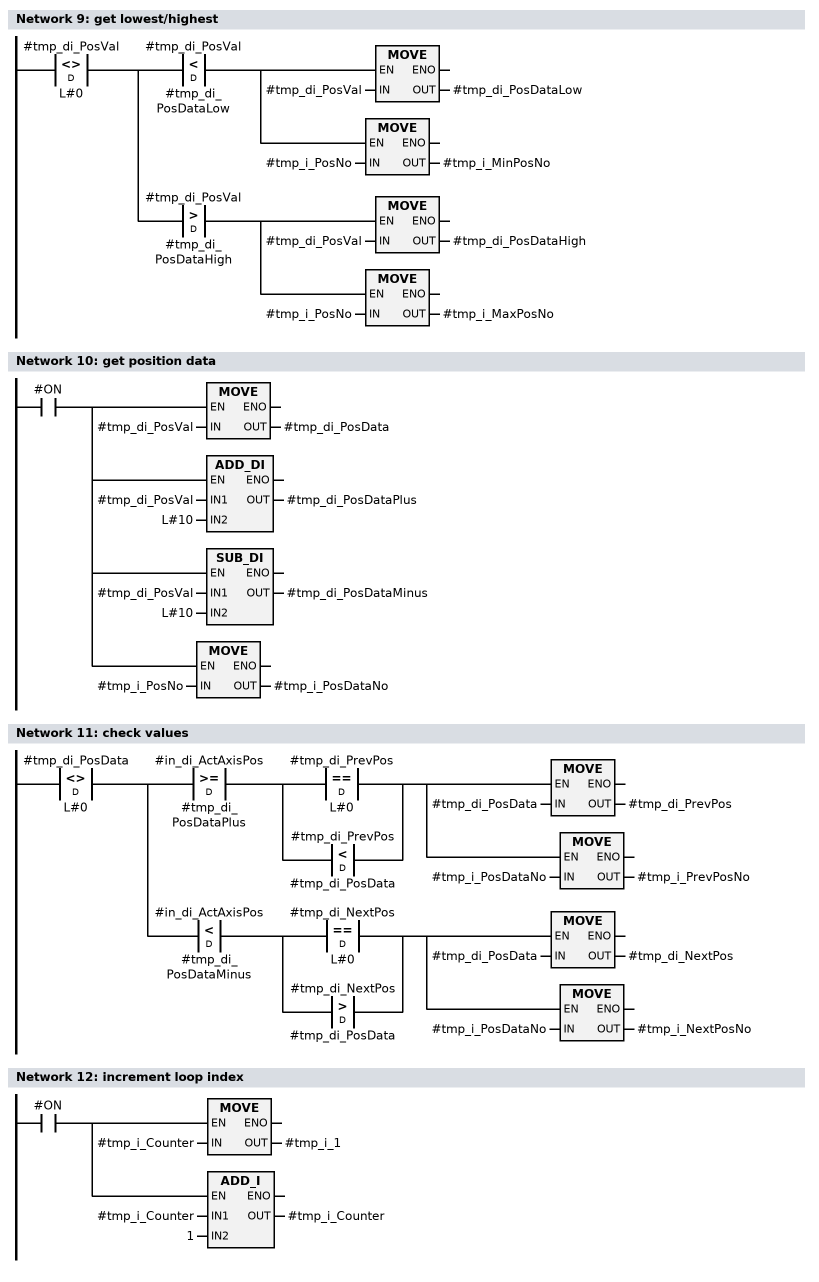
NETWORK
TITLE = get lowest/highest
      L     #tmp_di_PosVal;
      L     L#0;
      <>D;
      =     L 70.0;
      A     L 70.0;
      A(;
      L     #tmp_di_PosVal;
      L     #tmp_di_PosDataLow;
      <D;
      );
      =     L 70.1;
      A     L 70.1;
      JNB   _011;
      L     #tmp_di_PosVal;
      T     #tmp_di_PosDataLow;
_011: NOP   0;
      A     L 70.1;
      JNB   _012;
      L     #tmp_i_PosNo;
      T     #tmp_i_MinPosNo;
_012: NOP   0;
      A     L 70.0;
      A(;
      L     #tmp_di_PosVal;
      L     #tmp_di_PosDataHigh;
      >D;
      );
      =     L 70.1;
      A     L 70.1;
      JNB   _013;
      L     #tmp_di_PosVal;
      T     #tmp_di_PosDataHigh;
_013: NOP   0;
      A     L 70.1;
      JNB   _014;
      L     #tmp_i_PosNo;
      T     #tmp_i_MaxPosNo;
_014: NOP   0;
NETWORK
TITLE = get position data
      A     #ON;
      =     L 70.0;
      A     L 70.0;
      JNB   _015;
      L     #tmp_di_PosVal;
      T     #tmp_di_PosData;
_015: NOP   0;
      A     L 70.0;
      JNB   _016;
      L     #tmp_di_PosVal;
      L     L#10;
      +D;
      T     #tmp_di_PosDataPlus;
_016: NOP   0;
      A     L 70.0;
      JNB   _017;
      L     #tmp_di_PosVal;
      L     L#10;
      -D;
      T     #tmp_di_PosDataMinus;
_017: NOP   0;
      A     L 70.0;
      JNB   _018;
      L     #tmp_i_PosNo;
      T     #tmp_i_PosDataNo;
_018: NOP   0;
NETWORK
TITLE = check values
      L     #tmp_di_PosData;
      L     L#0;
      <>D;
      =     L 70.0;
      A     L 70.0;
      A(;
      L     #in_di_ActAxisPos;
      L     #tmp_di_PosDataPlus;
      >=D;
      );
      A(;
      O(;
      L     #tmp_di_PrevPos;
      L     L#0;
      ==D;
      );
      O(;
      L     #tmp_di_PrevPos;
      L     #tmp_di_PosData;
      <D;
      );
      );
      =     L 70.1;
      A     L 70.1;
      JNB   _019;
      L     #tmp_di_PosData;
      T     #tmp_di_PrevPos;
_019: NOP   0;
      A     L 70.1;
      JNB   _01a;
      L     #tmp_i_PosDataNo;
      T     #tmp_i_PrevPosNo;
_01a: NOP   0;
      A     L 70.0;
      A(;
      L     #in_di_ActAxisPos;
      L     #tmp_di_PosDataMinus;
      <D;
      );
      A(;
      O(;
      L     #tmp_di_NextPos;
      L     L#0;
      ==D;
      );
      O(;
      L     #tmp_di_NextPos;
      L     #tmp_di_PosData;
      >D;
      );
      );
      =     L 70.1;
      A     L 70.1;
      JNB   _01b;
      L     #tmp_di_PosData;
      T     #tmp_di_NextPos;
_01b: NOP   0;
      A     L 70.1;
      JNB   _01c;
      L     #tmp_i_PosDataNo;
      T     #tmp_i_NextPosNo;
_01c: NOP   0;
NETWORK
TITLE = increment loop index
      A     #ON;
      =     L 70.0;
      A     L 70.0;
      JNB   _01d;
      L     #tmp_i_Counter;
      T     #tmp_i_1;
_01d: NOP   0;
      A     L 70.0;
      JNB   _01e;
      L     #tmp_i_Counter;
      L     1;
      +I;
      T     #tmp_i_Counter;
_01e: NOP   0;
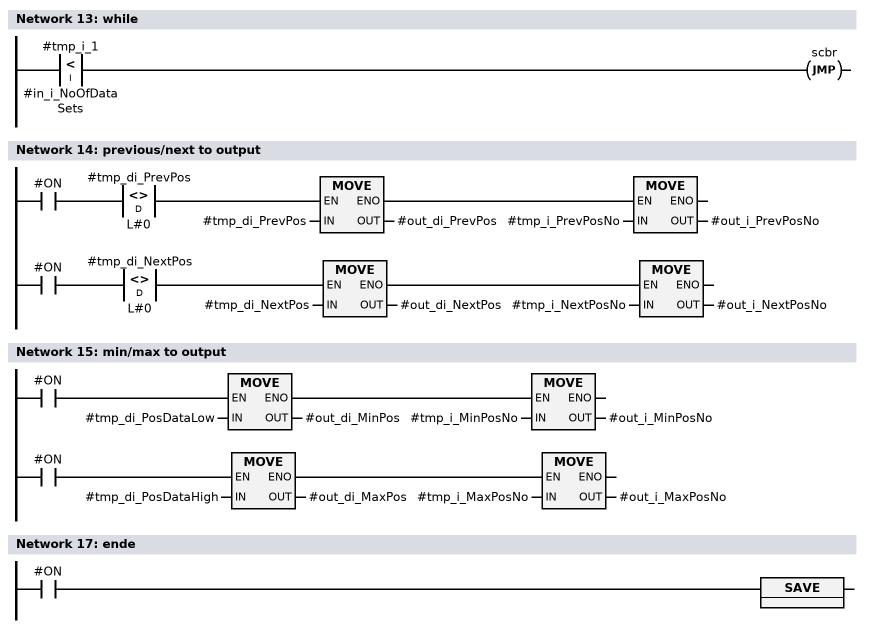
NETWORK
TITLE = while 
      L     #tmp_i_1;
      L     #in_i_NoOfDataSets;
      <I;
      JC    scbr;
NETWORK
TITLE = previous/next to output
      A     #ON;
      =     L 70.0;
      A(;
      A     L 70.0;
      A(;
      L     #tmp_di_PrevPos;
      L     L#0;
      <>D;
      );
      JNB   _01f;
      L     #tmp_di_PrevPos;
      T     #out_di_PrevPos;
      SET;
      SAVE;
      CLR;
_01f: A     BR;
      );
      JNB   _020;
      L     #tmp_i_PrevPosNo;
      T     #out_i_PrevPosNo;
_020: NOP   0;
      A(;
      A     L 70.0;
      A(;
      L     #tmp_di_NextPos;
      L     L#0;
      <>D;
      );
      JNB   _021;
      L     #tmp_di_NextPos;
      T     #out_di_NextPos;
      SET;
      SAVE;
      CLR;
_021: A     BR;
      );
      JNB   _022;
      L     #tmp_i_NextPosNo;
      T     #out_i_NextPosNo;
_022: NOP   0;
NETWORK
TITLE = min/max to output
      A     #ON;
      =     L 70.0;
      A(;
      A     L 70.0;
      JNB   _023;
      L     #tmp_di_PosDataLow;
      T     #out_di_MinPos;
      SET;
      SAVE;
      CLR;
_023: A     BR;
      );
      JNB   _024;
      L     #tmp_i_MinPosNo;
      T     #out_i_MinPosNo;
_024: NOP   0;
      A(;
      A     L 70.0;
      JNB   _025;
      L     #tmp_di_PosDataHigh;
      T     #out_di_MaxPos;
      SET;
      SAVE;
      CLR;
_025: A     BR;
      );
      JNB   _026;
      L     #tmp_i_MaxPosNo;
      T     #out_i_MaxPosNo;
_026: NOP   0;
NETWORK
TITLE = restore register
      LAR1  #Save_AR1;
      LAR2  #Save_AR2;
NETWORK
TITLE = ende
      A     #ON;
      SAVE;
END_FUNCTION

FUNCTION "Scan_BRI_DBs" : VOID	// FC 23
VERSION : 0.1
VAR_INPUT
  in_i_DBNo : INT ;
  in_i_ActRow : INT ;
  in_i_NoOfDataSets : INT ;
  in_di_DatSetLenght : DINT ;
  in_di_DataStartByte : DINT ;
  in_i_PosNo : INT ;
END_VAR
VAR_OUTPUT
  out_i_LIF_DBNo : INT ;
  out_i_LIF_DBNo_2 : INT ;
END_VAR
VAR_TEMP
  Save_AR1 : DWORD ;
  Save_AR2 : DWORD ;
  tmp_di_Pointer : DINT ;
  tmp_di_PosNo : DINT ;
  tmp_i_PosNo : INT ;
  tmp_i_ChkNo : INT ;
  tmp_i_DBNo : INT ;
  tmp_i_LIF_DBNo : INT ;
  tmp_i_LIF_DBNo_2 : INT ;
  tmp_i_offsetPointer : INT ;
  ON : BOOL ;
  tmp_b_LoopBrake : BOOL ;
  err_input : BOOL ;
END_VAR
BEGIN
NETWORK
TITLE = save register
      TAR1  #Save_AR1;
      TAR2  #Save_AR2;
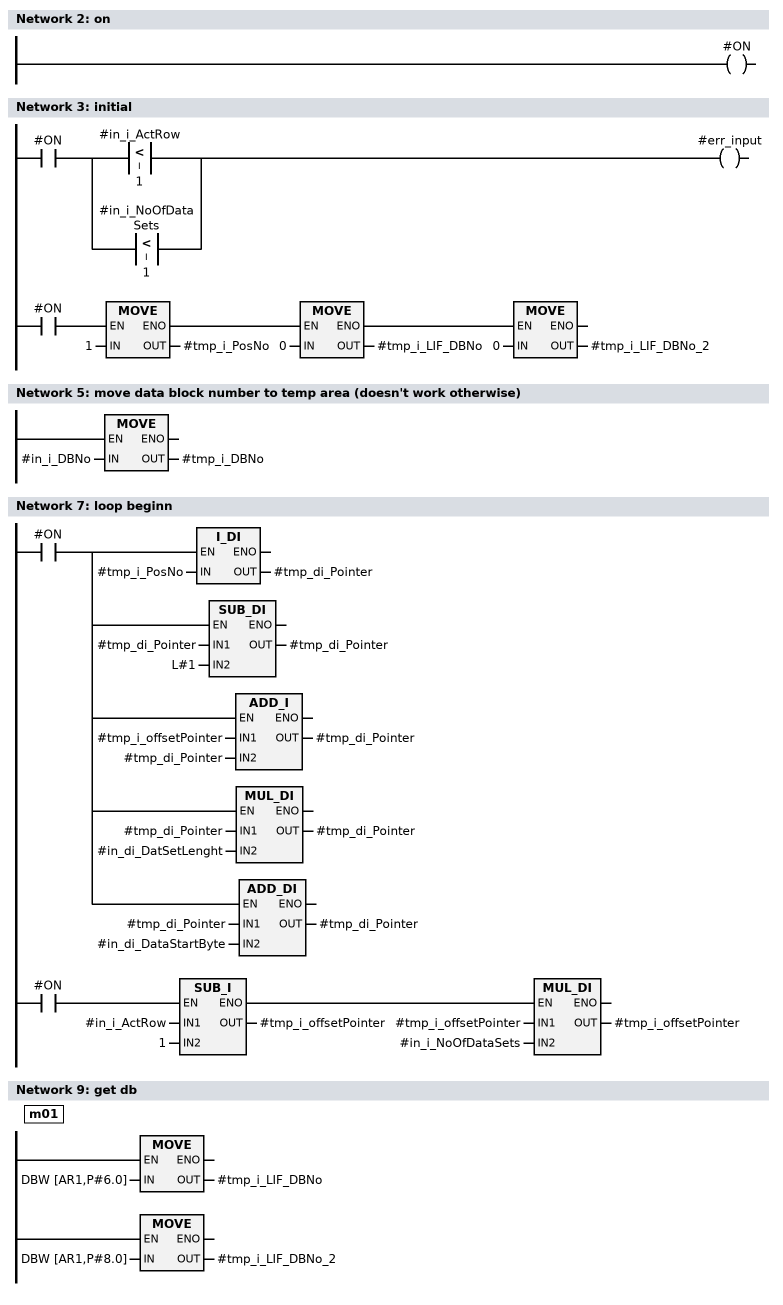
NETWORK
TITLE = on
      SET;
      =     #ON;
NETWORK
TITLE = initial
      A     #ON;
      =     L 30.0;
      A(;
      A(;
      A     L 30.0;
      JNB   _001;
      L     1;
      T     #tmp_i_PosNo;
      SET;
      SAVE;
      CLR;
_001: A     BR;
      );
      JNB   _002;
      L     0;
      T     #tmp_i_LIF_DBNo;
      SET;
      SAVE;
      CLR;
_002: A     BR;
      );
      JNB   _003;
      L     0;
      T     #tmp_i_LIF_DBNo_2;
_003: NOP   0;
      A     L 30.0;
      A(;
      O(;
      L     #in_i_ActRow;
      L     1;
      <I;
      );
      O(;
      L     #in_i_NoOfDataSets;
      L     1;
      <I;
      );
      );
      =     #err_input;
NETWORK
TITLE =
      AN    #err_input;
      JC    NoEr;	// On Error CLR all Outputs
      L     0;
      T     #out_i_LIF_DBNo;
      T     #out_i_LIF_DBNo_2;
      BEU;
NoEr: NOP   0;
NETWORK
TITLE = move data block number to temp area (doesn't work otherwise)
//doesn't work otherwise
      L     #in_i_DBNo;
      T     #tmp_i_DBNo;
      NOP   0;
NETWORK
TITLE = open DB
      OPN   DB [#tmp_i_DBNo];
NETWORK
TITLE = loop beginn
//calculate pointer to positionvalue
scbr: A     #ON;
      =     L 29.0;
      A     L 29.0;
      JNB   _008;
      L     #tmp_i_PosNo;
      ITD;
      T     #tmp_di_Pointer;
_008: NOP   0;
      A     L 29.0;
      JNB   _009;
      L     #tmp_di_Pointer;
      L     L#1;
      -D;
      T     #tmp_di_Pointer;
_009: NOP   0;
      A(;
      A     L 29.0;
      JNB   _00a;
      L     #in_i_ActRow;
      L     1;
      -I;
      T     #tmp_i_offsetPointer;
      AN    OV;
      SAVE;
      CLR;
_00a: A     BR;
      );
      JNB   _00b;
      L     #tmp_i_offsetPointer;
      L     #in_i_NoOfDataSets;
      *D;
      T     #tmp_i_offsetPointer;
_00b: NOP   0;
      A     L 29.0;
      JNB   _00c;
      L     #tmp_i_offsetPointer;
      L     #tmp_di_Pointer;
      +I;
      T     #tmp_di_Pointer;
_00c: NOP   0;
      A     L 29.0;
      JNB   _00d;
      L     #tmp_di_Pointer;
      L     #in_di_DatSetLenght;
      *D;
      T     #tmp_di_Pointer;
_00d: NOP   0;
      A     L 29.0;
      JNB   _00e;
      L     #tmp_di_Pointer;
      L     #in_di_DataStartByte;
      +D;
      T     #tmp_di_Pointer;
_00e: NOP   0;
NETWORK
TITLE = get position
      L     #tmp_di_Pointer;	// load pointer
      SLD   3;	// shift left 3 bits to achieve pointer format
      LAR1;	// load adressregister 1 with pointer
      L     DBW [AR1,P#0.0];	// load position number from DataBlock
      T     #tmp_i_ChkNo;	// Transfer to temp
      L     #tmp_i_ChkNo;
      L     #in_i_PosNo;
      ==I;
      JC    m01;
      L     #tmp_i_PosNo;
      L     1;
      +I;
      T     #tmp_i_PosNo;
      L     L#0;
      T     #tmp_di_PosNo;
      L     #tmp_i_PosNo;
      T     #tmp_di_PosNo;
      L     #tmp_di_PosNo;
      L     #in_i_NoOfDataSets;
      <=D;
      JC    scbr;
      JU    ende;
NETWORK
TITLE = get db
m01:  NOP   0;
      L     DBW [AR1,P#6.0];
      T     #tmp_i_LIF_DBNo;
      L     DBW [AR1,P#8.0];
      T     #tmp_i_LIF_DBNo_2;
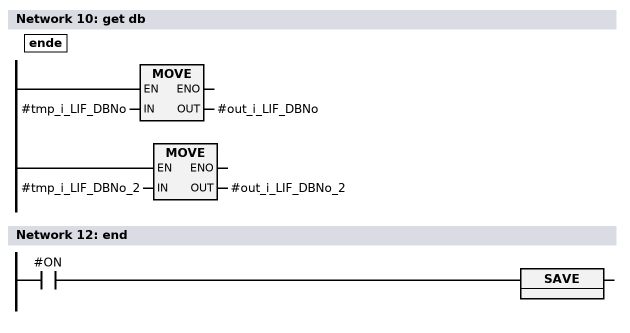
NETWORK
TITLE = get db
ende: NOP   0;
      L     #tmp_i_LIF_DBNo;
      T     #out_i_LIF_DBNo;
      L     #tmp_i_LIF_DBNo_2;
      T     #out_i_LIF_DBNo_2;
NETWORK
TITLE = restore register
      LAR1  #Save_AR1;
      LAR2  #Save_AR2;
NETWORK
TITLE = end
      A     #ON;
      SAVE;
END_FUNCTION

FUNCTION "Scan_LIF" : VOID	// FC 25
TITLE = scan positions lift
VERSION : 1.0
VAR_INPUT
  in_x_ReleaseScan : BOOL ;
  in_i_LiDbNo : INT ;
  in_di_NoOfDataSetsli : DINT ;
  in_di_DatSetLenghtli : DINT ;
  in_di_ActAxisPos : DINT ;
  in_di_AreaWin : DINT ;
  in_di_PosWin : DINT ;
END_VAR
VAR_OUTPUT
  out_di_Pointer : DINT ;
  out_i_AreaNo : INT ;
  out_b_InArea : BOOL ;
  out_b_InPosHo : BOOL ;
  out_b_InPosHu : BOOL ;
  out_di_PosValHo : DINT ;
  out_di_PosValHu : DINT ;
  out_HookDataSet : UDT 102;
END_VAR
VAR_TEMP
  tmp_any_1 : ANY ;
  tmp_di_Pointer : DINT ;
  tmp_di_PosWinMinus : DINT ;
  tmp_di_PosWinPlus : DINT ;
  tmp_di_1 : DINT ;
  tmp_di_PosValHu : DINT ;
  tmp_i_PosNo : INT ;
  tmp_i_Hooktype : INT ;
  tmp_i_DbNo : INT ;
  ON : BOOL ;
  OFF : BOOL ;
  tmp_b_LoopBrake : BOOL ;
  tmp_b_1 : BOOL ;
  Save_AR1 : DWORD ;
  Save_AR2 : DWORD ;
  RetVal : INT ;
  tmpHookDataSet : UDT 102;
END_VAR
BEGIN
NETWORK
TITLE = save register
      TAR1  #Save_AR1;
      TAR2  #Save_AR2;
NETWORK
TITLE = on/off
      SET;
      =     #ON;
      CLR;
      =     #OFF;
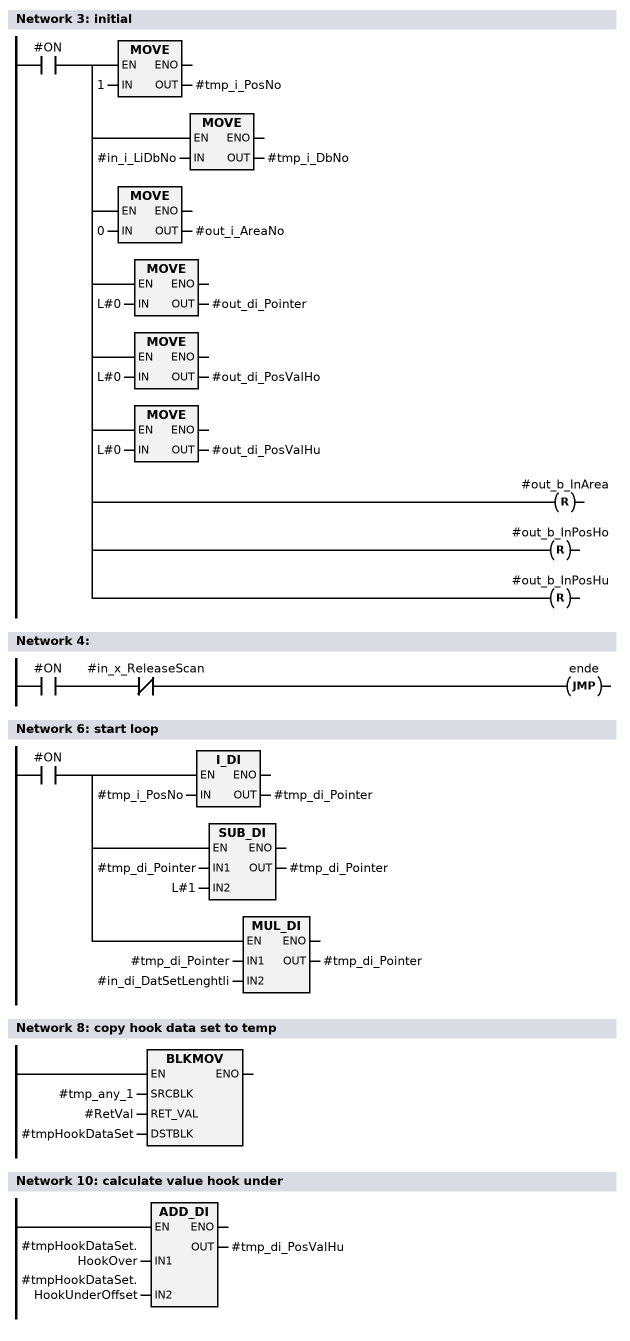
NETWORK
TITLE = initial
//#in_DbNo -> #tmp.. while "AUF DB" only with #tmp...
      A     #ON;
      =     L 104.0;
      A     L 104.0;
      JNB   _001;
      L     1;
      T     #tmp_i_PosNo;
_001: NOP   0;
      A     L 104.0;
      JNB   _002;
      L     #in_i_LiDbNo;
      T     #tmp_i_DbNo;
_002: NOP   0;
      A     L 104.0;
      JNB   _003;
      L     0;
      T     #out_i_AreaNo;
_003: NOP   0;
      A     L 104.0;
      JNB   _004;
      L     L#0;
      T     #out_di_Pointer;
_004: NOP   0;
      A     L 104.0;
      JNB   _005;
      L     L#0;
      T     #out_di_PosValHo;
_005: NOP   0;
      A     L 104.0;
      JNB   _006;
      L     L#0;
      T     #out_di_PosValHu;
_006: NOP   0;
      A     L 104.0;
      BLD   102;
      R     #out_b_InArea;
      A     L 104.0;
      BLD   102;
      R     #out_b_InPosHo;
      A     L 104.0;
      BLD   102;
      R     #out_b_InPosHu;
NETWORK
TITLE =
      A     #ON;
      AN    #in_x_ReleaseScan;
      JC    ende;
NETWORK
TITLE = open DB/DI
      OPN   DB [#tmp_i_DbNo];
NETWORK
TITLE = start loop
//calculate Pointer to dataset
scli: A     #ON;
      =     L 104.0;
      A     L 104.0;
      JNB   _007;
      L     #tmp_i_PosNo;
      ITD;
      T     #tmp_di_Pointer;
_007: NOP   0;
      A     L 104.0;
      JNB   _008;
      L     #tmp_di_Pointer;
      L     L#1;
      -D;
      T     #tmp_di_Pointer;
_008: NOP   0;
      A     L 104.0;
      JNB   _009;
      L     #tmp_di_Pointer;
      L     #in_di_DatSetLenghtli;
      *D;
      T     #tmp_di_Pointer;
_009: NOP   0;
NETWORK
TITLE = create any-pointer to hookdataset
      L     W#16#1002;
      T     LW 0;
      L     56;
      T     LW 2;
      L     #tmp_i_DbNo;
      T     LW 4;
      L     #tmp_di_Pointer;
      SLD   3;
      OD    DW#16#84000000;
      T     LD 6;
NETWORK
TITLE = copy hook data set to temp
      CALL  "BLKMOV" (
           SRCBLK                   := #tmp_any_1,
           RET_VAL                  := #RetVal,
           DSTBLK                   := #tmpHookDataSet);
      NOP   0;
NETWORK
TITLE = copy hook data to out
      A     #ON;
      =     L 104.0;
      A(;
      A     L 104.0;
      JNB   _00a;
      L     #tmpHookDataSet.HookOver;
      BLD   5;
      T     LD 107;
      TAK;
      T     LD 111;
      L     P##out_HookDataSet;
      LAR1;
      L     W [AR1,P#0.0];
      T     LW 105;
      OPN   DB [LW 105];
      L     D [AR1,P#2.0];
      LAR1;
      L     LD 111;
      L     LD 107;
      T     D [AR1,P#0.0];
      SET;
      SAVE;
      CLR;
_00a: A     BR;
      );
      JNB   _00b;
      L     #tmpHookDataSet.HookUnderOffset;
      BLD   5;
      T     LD 107;
      TAK;
      T     LD 111;
      L     P##out_HookDataSet;
      LAR1;
      L     W [AR1,P#0.0];
      T     LW 105;
      OPN   DB [LW 105];
      L     D [AR1,P#2.0];
      LAR1;
      L     LD 111;
      L     LD 107;
      T     D [AR1,P#4.0];
_00b: NOP   0;
      A(;
      A(;
      A     L 104.0;
      JNB   _00c;
      L     #tmpHookDataSet.TelPos_1.TelPos;
      BLD   5;
      T     LD 107;
      TAK;
      T     LD 111;
      L     P##out_HookDataSet;
      LAR1;
      L     W [AR1,P#0.0];
      T     LW 105;
      OPN   DB [LW 105];
      L     D [AR1,P#2.0];
      LAR1;
      L     LD 111;
      L     LD 107;
      T     D [AR1,P#18.0];
      SET;
      SAVE;
      CLR;
_00c: A     BR;
      );
      JNB   _00d;
      L     #tmpHookDataSet.TelPos_2.TelPos;
      BLD   5;
      T     LD 107;
      TAK;
      T     LD 111;
      L     P##out_HookDataSet;
      LAR1;
      L     W [AR1,P#0.0];
      T     LW 105;
      OPN   DB [LW 105];
      L     D [AR1,P#2.0];
      LAR1;
      L     LD 111;
      L     LD 107;
      T     D [AR1,P#34.0];
      SET;
      SAVE;
      CLR;
_00d: A     BR;
      );
      JNB   _00e;
      L     #tmpHookDataSet.TelPos_3.TelPos;
      BLD   5;
      T     LD 107;
      TAK;
      T     LD 111;
      L     P##out_HookDataSet;
      LAR1;
      L     W [AR1,P#0.0];
      T     LW 105;
      OPN   DB [LW 105];
      L     D [AR1,P#2.0];
      LAR1;
      L     LD 111;
      L     LD 107;
      T     D [AR1,P#50.0];
_00e: NOP   0;
      A(;
      A(;
      A     L 104.0;
      JNB   _00f;
      L     #tmpHookDataSet.TelPos_1.TotLengthMin;
      BLD   5;
      T     LD 107;
      TAK;
      T     LD 111;
      L     P##out_HookDataSet;
      LAR1;
      L     W [AR1,P#0.0];
      T     LW 105;
      OPN   DB [LW 105];
      L     D [AR1,P#2.0];
      LAR1;
      L     LD 111;
      L     LD 107;
      T     W [AR1,P#10.0];
      SET;
      SAVE;
      CLR;
_00f: A     BR;
      );
      JNB   _010;
      L     #tmpHookDataSet.TelPos_1.TotLengthMax;
      BLD   5;
      T     LD 107;
      TAK;
      T     LD 111;
      L     P##out_HookDataSet;
      LAR1;
      L     W [AR1,P#0.0];
      T     LW 105;
      OPN   DB [LW 105];
      L     D [AR1,P#2.0];
      LAR1;
      L     LD 111;
      L     LD 107;
      T     W [AR1,P#12.0];
      SET;
      SAVE;
      CLR;
_010: A     BR;
      );
      JNB   _011;
      L     #tmpHookDataSet.TelPos_1.FaceLengthMax;
      BLD   5;
      T     LD 107;
      TAK;
      T     LD 111;
      L     P##out_HookDataSet;
      LAR1;
      L     W [AR1,P#0.0];
      T     LW 105;
      OPN   DB [LW 105];
      L     D [AR1,P#2.0];
      LAR1;
      L     LD 111;
      L     LD 107;
      T     W [AR1,P#14.0];
_011: NOP   0;
      A(;
      A(;
      A     L 104.0;
      JNB   _012;
      L     #tmpHookDataSet.TelPos_1.CircumMax;
      BLD   5;
      T     LD 107;
      TAK;
      T     LD 111;
      L     P##out_HookDataSet;
      LAR1;
      L     W [AR1,P#0.0];
      T     LW 105;
      OPN   DB [LW 105];
      L     D [AR1,P#2.0];
      LAR1;
      L     LD 111;
      L     LD 107;
      T     W [AR1,P#16.0];
      SET;
      SAVE;
      CLR;
_012: A     BR;
      );
      JNB   _013;
      L     #tmpHookDataSet.TelPos_1.HookType;
      BLD   5;
      T     LD 107;
      TAK;
      T     LD 111;
      L     P##out_HookDataSet;
      LAR1;
      L     W [AR1,P#0.0];
      T     LW 105;
      OPN   DB [LW 105];
      L     D [AR1,P#2.0];
      LAR1;
      L     LD 111;
      L     LD 107;
      T     W [AR1,P#8.0];
      SET;
      SAVE;
      CLR;
_013: A     BR;
      );
      JNB   _014;
      L     #tmpHookDataSet.TelPos_1.Reserve1;
      BLD   5;
      T     LD 107;
      TAK;
      T     LD 111;
      L     P##out_HookDataSet;
      LAR1;
      L     W [AR1,P#0.0];
      T     LW 105;
      OPN   DB [LW 105];
      L     D [AR1,P#2.0];
      LAR1;
      L     LD 111;
      L     LD 107;
      T     W [AR1,P#22.0];
_014: NOP   0;
      A(;
      A(;
      A     L 104.0;
      JNB   _015;
      L     #tmpHookDataSet.TelPos_2.TotLengthMin;
      BLD   5;
      T     LD 107;
      TAK;
      T     LD 111;
      L     P##out_HookDataSet;
      LAR1;
      L     W [AR1,P#0.0];
      T     LW 105;
      OPN   DB [LW 105];
      L     D [AR1,P#2.0];
      LAR1;
      L     LD 111;
      L     LD 107;
      T     W [AR1,P#26.0];
      SET;
      SAVE;
      CLR;
_015: A     BR;
      );
      JNB   _016;
      L     #tmpHookDataSet.TelPos_2.TotLengthMax;
      BLD   5;
      T     LD 107;
      TAK;
      T     LD 111;
      L     P##out_HookDataSet;
      LAR1;
      L     W [AR1,P#0.0];
      T     LW 105;
      OPN   DB [LW 105];
      L     D [AR1,P#2.0];
      LAR1;
      L     LD 111;
      L     LD 107;
      T     W [AR1,P#28.0];
      SET;
      SAVE;
      CLR;
_016: A     BR;
      );
      JNB   _017;
      L     #tmpHookDataSet.TelPos_2.FaceLengthMax;
      BLD   5;
      T     LD 107;
      TAK;
      T     LD 111;
      L     P##out_HookDataSet;
      LAR1;
      L     W [AR1,P#0.0];
      T     LW 105;
      OPN   DB [LW 105];
      L     D [AR1,P#2.0];
      LAR1;
      L     LD 111;
      L     LD 107;
      T     W [AR1,P#30.0];
_017: NOP   0;
      A(;
      A(;
      A     L 104.0;
      JNB   _018;
      L     #tmpHookDataSet.TelPos_2.CircumMax;
      BLD   5;
      T     LD 107;
      TAK;
      T     LD 111;
      L     P##out_HookDataSet;
      LAR1;
      L     W [AR1,P#0.0];
      T     LW 105;
      OPN   DB [LW 105];
      L     D [AR1,P#2.0];
      LAR1;
      L     LD 111;
      L     LD 107;
      T     W [AR1,P#32.0];
      SET;
      SAVE;
      CLR;
_018: A     BR;
      );
      JNB   _019;
      L     #tmpHookDataSet.TelPos_2.HookType;
      BLD   5;
      T     LD 107;
      TAK;
      T     LD 111;
      L     P##out_HookDataSet;
      LAR1;
      L     W [AR1,P#0.0];
      T     LW 105;
      OPN   DB [LW 105];
      L     D [AR1,P#2.0];
      LAR1;
      L     LD 111;
      L     LD 107;
      T     W [AR1,P#24.0];
      SET;
      SAVE;
      CLR;
_019: A     BR;
      );
      JNB   _01a;
      L     #tmpHookDataSet.TelPos_2.Reserve1;
      BLD   5;
      T     LD 107;
      TAK;
      T     LD 111;
      L     P##out_HookDataSet;
      LAR1;
      L     W [AR1,P#0.0];
      T     LW 105;
      OPN   DB [LW 105];
      L     D [AR1,P#2.0];
      LAR1;
      L     LD 111;
      L     LD 107;
      T     W [AR1,P#38.0];
_01a: NOP   0;
      A(;
      A(;
      A     L 104.0;
      JNB   _01b;
      L     #tmpHookDataSet.TelPos_3.TotLengthMin;
      BLD   5;
      T     LD 107;
      TAK;
      T     LD 111;
      L     P##out_HookDataSet;
      LAR1;
      L     W [AR1,P#0.0];
      T     LW 105;
      OPN   DB [LW 105];
      L     D [AR1,P#2.0];
      LAR1;
      L     LD 111;
      L     LD 107;
      T     W [AR1,P#42.0];
      SET;
      SAVE;
      CLR;
_01b: A     BR;
      );
      JNB   _01c;
      L     #tmpHookDataSet.TelPos_3.TotLengthMax;
      BLD   5;
      T     LD 107;
      TAK;
      T     LD 111;
      L     P##out_HookDataSet;
      LAR1;
      L     W [AR1,P#0.0];
      T     LW 105;
      OPN   DB [LW 105];
      L     D [AR1,P#2.0];
      LAR1;
      L     LD 111;
      L     LD 107;
      T     W [AR1,P#44.0];
      SET;
      SAVE;
      CLR;
_01c: A     BR;
      );
      JNB   _01d;
      L     #tmpHookDataSet.TelPos_3.FaceLengthMax;
      BLD   5;
      T     LD 107;
      TAK;
      T     LD 111;
      L     P##out_HookDataSet;
      LAR1;
      L     W [AR1,P#0.0];
      T     LW 105;
      OPN   DB [LW 105];
      L     D [AR1,P#2.0];
      LAR1;
      L     LD 111;
      L     LD 107;
      T     W [AR1,P#46.0];
_01d: NOP   0;
      A(;
      A(;
      A     L 104.0;
      JNB   _01e;
      L     #tmpHookDataSet.TelPos_3.CircumMax;
      BLD   5;
      T     LD 107;
      TAK;
      T     LD 111;
      L     P##out_HookDataSet;
      LAR1;
      L     W [AR1,P#0.0];
      T     LW 105;
      OPN   DB [LW 105];
      L     D [AR1,P#2.0];
      LAR1;
      L     LD 111;
      L     LD 107;
      T     W [AR1,P#48.0];
      SET;
      SAVE;
      CLR;
_01e: A     BR;
      );
      JNB   _01f;
      L     #tmpHookDataSet.TelPos_3.HookType;
      BLD   5;
      T     LD 107;
      TAK;
      T     LD 111;
      L     P##out_HookDataSet;
      LAR1;
      L     W [AR1,P#0.0];
      T     LW 105;
      OPN   DB [LW 105];
      L     D [AR1,P#2.0];
      LAR1;
      L     LD 111;
      L     LD 107;
      T     W [AR1,P#40.0];
      SET;
      SAVE;
      CLR;
_01f: A     BR;
      );
      JNB   _020;
      L     #tmpHookDataSet.TelPos_3.Reserve1;
      BLD   5;
      T     LD 107;
      TAK;
      T     LD 111;
      L     P##out_HookDataSet;
      LAR1;
      L     W [AR1,P#0.0];
      T     LW 105;
      OPN   DB [LW 105];
      L     D [AR1,P#2.0];
      LAR1;
      L     LD 111;
      L     LD 107;
      T     W [AR1,P#54.0];
_020: NOP   0;
NETWORK
TITLE = calculate value hook under
      L     #tmpHookDataSet.HookOver;
      L     #tmpHookDataSet.HookUnderOffset;
      +D;
      T     #tmp_di_PosValHu;
      NOP   0;
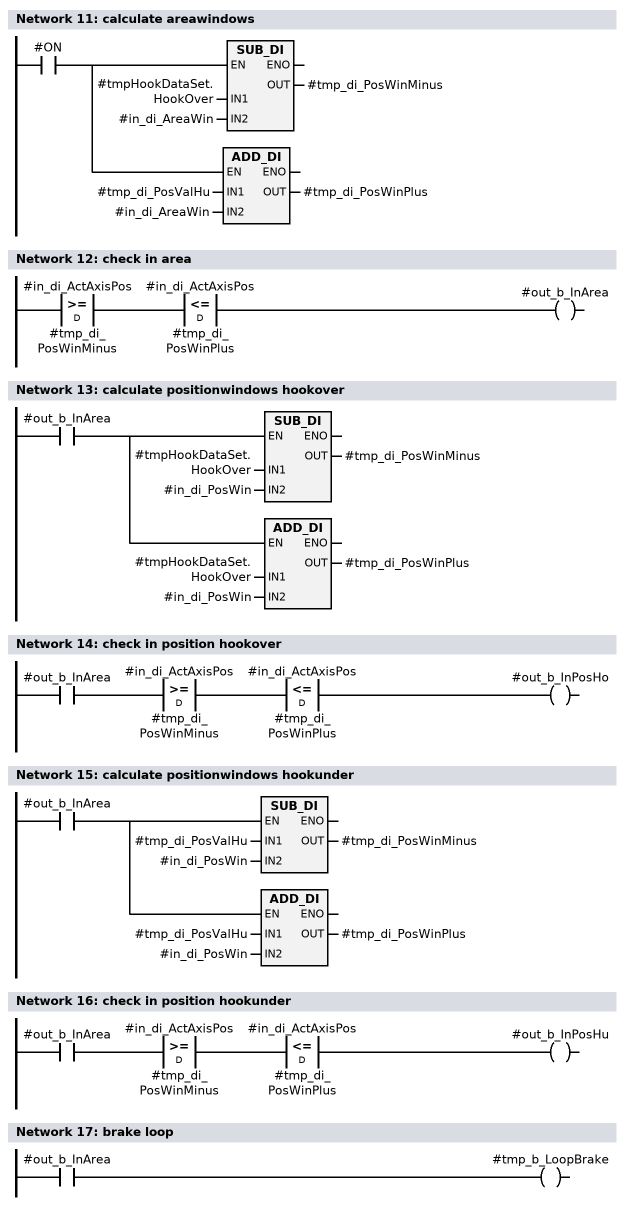
NETWORK
TITLE = calculate areawindows
      A     #ON;
      =     L 104.0;
      A     L 104.0;
      JNB   _021;
      L     #tmpHookDataSet.HookOver;
      L     #in_di_AreaWin;
      -D;
      T     #tmp_di_PosWinMinus;
_021: NOP   0;
      A     L 104.0;
      JNB   _022;
      L     #tmp_di_PosValHu;
      L     #in_di_AreaWin;
      +D;
      T     #tmp_di_PosWinPlus;
_022: NOP   0;
NETWORK
TITLE = check in area
      A(;
      L     #in_di_ActAxisPos;
      L     #tmp_di_PosWinMinus;
      >=D;
      );
      A(;
      L     #in_di_ActAxisPos;
      L     #tmp_di_PosWinPlus;
      <=D;
      );
      =     #out_b_InArea;
NETWORK
TITLE = calculate positionwindows hookover
      A     #out_b_InArea;
      =     L 104.0;
      A     L 104.0;
      JNB   _023;
      L     #tmpHookDataSet.HookOver;
      L     #in_di_PosWin;
      -D;
      T     #tmp_di_PosWinMinus;
_023: NOP   0;
      A     L 104.0;
      JNB   _024;
      L     #tmpHookDataSet.HookOver;
      L     #in_di_PosWin;
      +D;
      T     #tmp_di_PosWinPlus;
_024: NOP   0;
NETWORK
TITLE = check in position hookover
      A     #out_b_InArea;
      A(;
      L     #in_di_ActAxisPos;
      L     #tmp_di_PosWinMinus;
      >=D;
      );
      A(;
      L     #in_di_ActAxisPos;
      L     #tmp_di_PosWinPlus;
      <=D;
      );
      =     #out_b_InPosHo;
NETWORK
TITLE = calculate positionwindows hookunder
      A     #out_b_InArea;
      =     L 104.0;
      A     L 104.0;
      JNB   _025;
      L     #tmp_di_PosValHu;
      L     #in_di_PosWin;
      -D;
      T     #tmp_di_PosWinMinus;
_025: NOP   0;
      A     L 104.0;
      JNB   _026;
      L     #tmp_di_PosValHu;
      L     #in_di_PosWin;
      +D;
      T     #tmp_di_PosWinPlus;
_026: NOP   0;
NETWORK
TITLE = check in position hookunder
      A     #out_b_InArea;
      A(;
      L     #in_di_ActAxisPos;
      L     #tmp_di_PosWinMinus;
      >=D;
      );
      A(;
      L     #in_di_ActAxisPos;
      L     #tmp_di_PosWinPlus;
      <=D;
      );
      =     #out_b_InPosHu;
NETWORK
TITLE = brake loop
      A     #out_b_InArea;
      =     #tmp_b_LoopBrake;
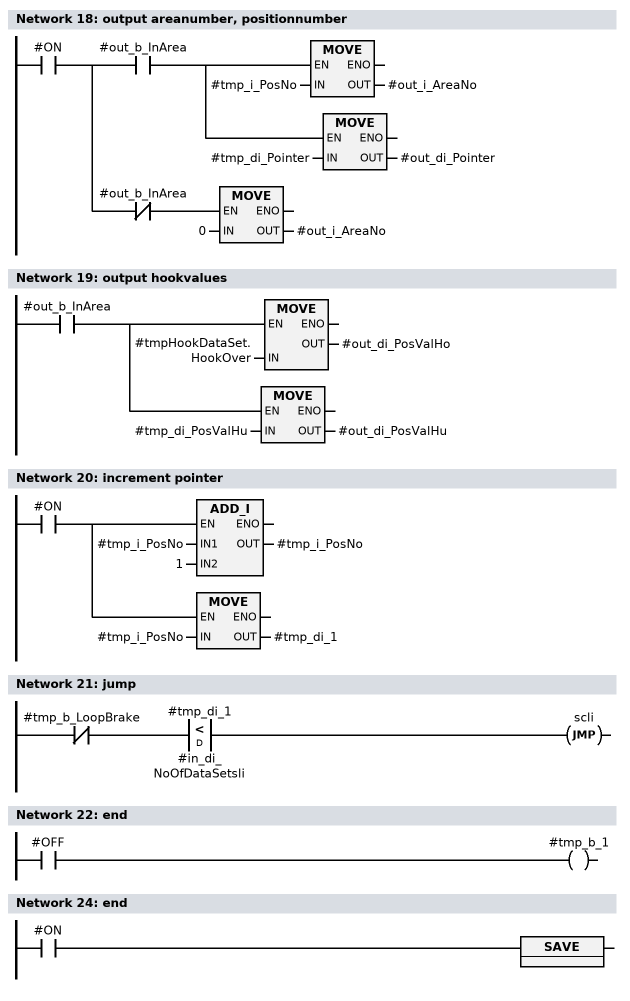
NETWORK
TITLE = output areanumber, positionnumber
      A     #ON;
      =     L 104.0;
      A     L 104.0;
      A     #out_b_InArea;
      =     L 104.1;
      A     L 104.1;
      JNB   _027;
      L     #tmp_i_PosNo;
      T     #out_i_AreaNo;
_027: NOP   0;
      A     L 104.1;
      JNB   _028;
      L     #tmp_di_Pointer;
      T     #out_di_Pointer;
_028: NOP   0;
      A     L 104.0;
      AN    #out_b_InArea;
      JNB   _029;
      L     0;
      T     #out_i_AreaNo;
_029: NOP   0;
NETWORK
TITLE = output hookvalues 
      A     #out_b_InArea;
      =     L 104.0;
      A     L 104.0;
      JNB   _02a;
      L     #tmpHookDataSet.HookOver;
      T     #out_di_PosValHo;
_02a: NOP   0;
      A     L 104.0;
      JNB   _02b;
      L     #tmp_di_PosValHu;
      T     #out_di_PosValHu;
_02b: NOP   0;
NETWORK
TITLE = increment pointer
      A     #ON;
      =     L 104.0;
      A     L 104.0;
      JNB   _02c;
      L     #tmp_i_PosNo;
      L     1;
      +I;
      T     #tmp_i_PosNo;
_02c: NOP   0;
      A     L 104.0;
      JNB   _02d;
      L     #tmp_i_PosNo;
      T     #tmp_di_1;
_02d: NOP   0;
NETWORK
TITLE = jump
      AN    #tmp_b_LoopBrake;
      A(;
      L     #tmp_di_1;
      L     #in_di_NoOfDataSetsli;
      <D;
      );
      JC    scli;
NETWORK
TITLE = end
ende: A     #OFF;
      =     #tmp_b_1;
NETWORK
TITLE = restore register
      LAR1  #Save_AR1;
      LAR2  #Save_AR2;
NETWORK
TITLE = end
      A     #ON;
      SAVE;
END_FUNCTION

FUNCTION "Scan_LIF_Man" : VOID	// FC 26
TITLE = scan positions LIFt manual mode
VERSION : 1.0
VAR_INPUT
  in_b_release : BOOL ;
  in_i_DBNo : INT ;
  in_i_NoOfDataSets : INT ;
  in_i_DatSetLenght : INT ;
  in_i_DataStartByte : INT ;
  in_di_ActAxisPos : DINT ;
  in_b_Free : BOOL ;
  in_b_Occupied : BOOL ;
END_VAR
VAR_OUTPUT
  out_di_PrevPos : DINT ;
  out_di_ActPos : DINT ;
  out_di_NextPos : DINT ;
  out_di_MinPos : DINT ;
  out_di_MaxPos : DINT ;
END_VAR
VAR_TEMP
  Save_AR1 : DWORD ;
  Save_AR2 : DWORD ;
  tmp_di_1 : DINT ;
  tmp_di_Pointer : DINT ;
  tmp_di_ChkPosValHo : DINT ;
  tmp_di_ChkPosValHu : DINT ;
  tmp_di_ChkPosVal : DINT ;
  tmp_di_PosData : DINT ;
  tmp_di_PosDataPlus : DINT ;
  tmp_di_PosDataMinus : DINT ;
  tmp_di_PosDataLow : DINT ;
  tmp_di_PosDataHigh : DINT ;
  tmp_di_PrevPos : DINT ;
  tmp_di_NextPos : DINT ;
  tmp_i_Counter : INT ;
  tmp_i_DBNo : INT ;
  tmp_i_NoOfDataSets : INT ;
  tmp_i : INT ;
  ON : BOOL ;
  OFF : BOOL ;
  tmp_b_1 : BOOL ;
END_VAR
BEGIN
NETWORK
TITLE = save register
      TAR1  #Save_AR1;
      TAR2  #Save_AR2;
NETWORK
TITLE = on/off
      SET;
      =     #ON;
      CLR;
      =     #OFF;
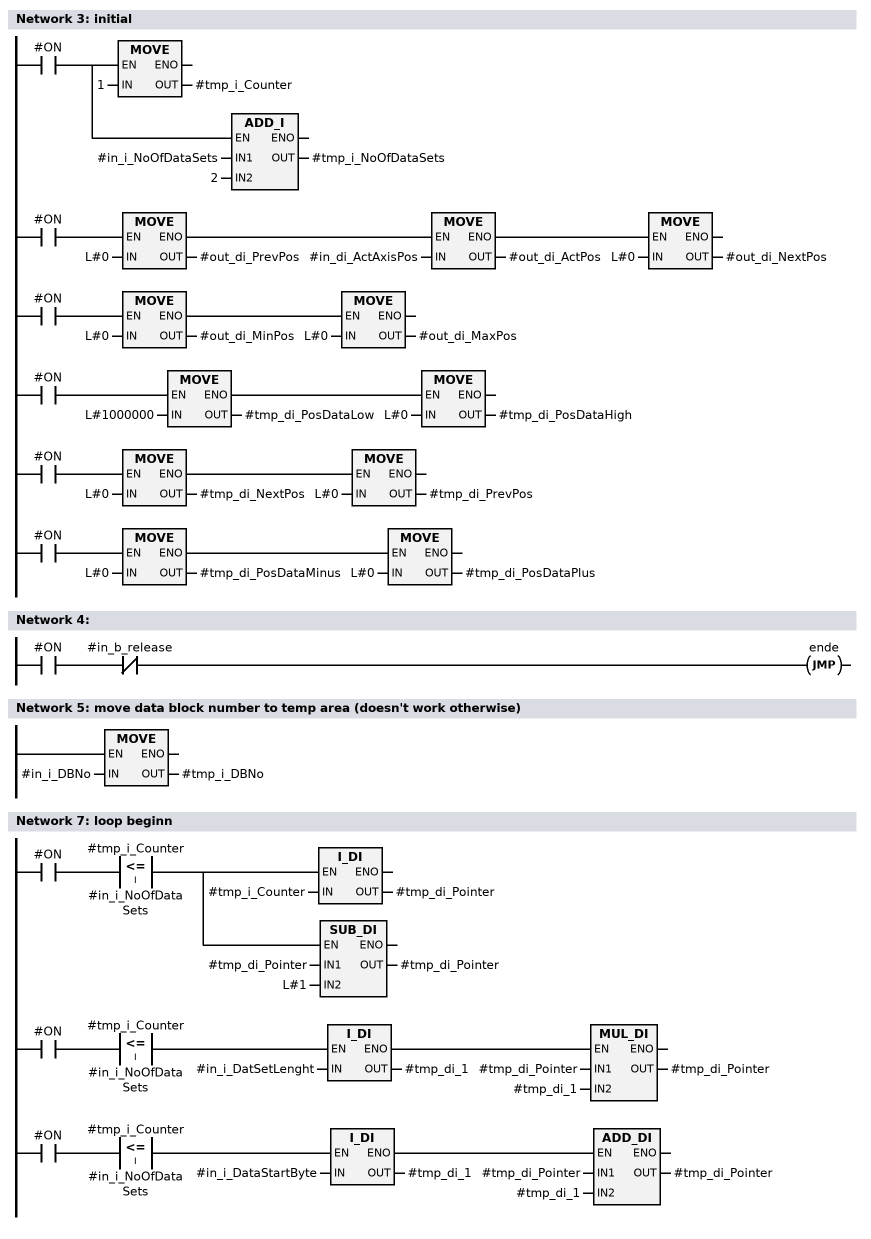
NETWORK
TITLE = initial
//set loopcounter to 0
//reset outputs
      A     #ON;
      =     L 65.0;
      A     L 65.0;
      JNB   _001;
      L     1;
      T     #tmp_i_Counter;
_001: NOP   0;
      A(;
      A(;
      A     L 65.0;
      JNB   _002;
      L     L#0;
      T     #out_di_PrevPos;
      SET;
      SAVE;
      CLR;
_002: A     BR;
      );
      JNB   _003;
      L     #in_di_ActAxisPos;
      T     #out_di_ActPos;
      SET;
      SAVE;
      CLR;
_003: A     BR;
      );
      JNB   _004;
      L     L#0;
      T     #out_di_NextPos;
_004: NOP   0;
      A(;
      A     L 65.0;
      JNB   _005;
      L     L#0;
      T     #out_di_MinPos;
      SET;
      SAVE;
      CLR;
_005: A     BR;
      );
      JNB   _006;
      L     L#0;
      T     #out_di_MaxPos;
_006: NOP   0;
      A(;
      A     L 65.0;
      JNB   _007;
      L     L#1000000;
      T     #tmp_di_PosDataLow;
      SET;
      SAVE;
      CLR;
_007: A     BR;
      );
      JNB   _008;
      L     L#0;
      T     #tmp_di_PosDataHigh;
_008: NOP   0;
      A(;
      A     L 65.0;
      JNB   _009;
      L     L#0;
      T     #tmp_di_NextPos;
      SET;
      SAVE;
      CLR;
_009: A     BR;
      );
      JNB   _00a;
      L     L#0;
      T     #tmp_di_PrevPos;
_00a: NOP   0;
      A(;
      A     L 65.0;
      JNB   _00b;
      L     L#0;
      T     #tmp_di_PosDataMinus;
      SET;
      SAVE;
      CLR;
_00b: A     BR;
      );
      JNB   _00c;
      L     L#0;
      T     #tmp_di_PosDataPlus;
_00c: NOP   0;
      A     L 65.0;
      JNB   _00d;
      L     #in_i_NoOfDataSets;
      L     2;
      +I;
      T     #tmp_i_NoOfDataSets;
_00d: NOP   0;
NETWORK
TITLE =
      A     #ON;
      AN    #in_b_release;
      JC    ende;
NETWORK
TITLE = move data block number to temp area (doesn't work otherwise)
//doesn't work otherwise
      L     #in_i_DBNo;
      T     #tmp_i_DBNo;
      NOP   0;
NETWORK
TITLE = open DB
      OPN   DB [#tmp_i_DBNo];
NETWORK
TITLE = loop beginn
//calculate pointer to positionvalue
scbr: A     #ON;
      A(;
      L     #tmp_i_Counter;
      L     #in_i_NoOfDataSets;
      <=I;
      );
      =     L 65.0;
      A     L 65.0;
      JNB   _00e;
      L     #tmp_i_Counter;
      ITD;
      T     #tmp_di_Pointer;
_00e: NOP   0;
      A     L 65.0;
      JNB   _00f;
      L     #tmp_di_Pointer;
      L     L#1;
      -D;
      T     #tmp_di_Pointer;
_00f: NOP   0;
      A(;
      A     L 65.0;
      JNB   _010;
      L     #in_i_DatSetLenght;
      ITD;
      T     #tmp_di_1;
      SET;
      SAVE;
      CLR;
_010: A     BR;
      );
      JNB   _011;
      L     #tmp_di_Pointer;
      L     #tmp_di_1;
      *D;
      T     #tmp_di_Pointer;
_011: NOP   0;
      A(;
      A     L 65.0;
      JNB   _012;
      L     #in_i_DataStartByte;
      ITD;
      T     #tmp_di_1;
      SET;
      SAVE;
      CLR;
_012: A     BR;
      );
      JNB   _013;
      L     #tmp_di_Pointer;
      L     #tmp_di_1;
      +D;
      T     #tmp_di_Pointer;
_013: NOP   0;
NETWORK
TITLE = get values from db-hooks
      L     #tmp_di_Pointer;	// load pointer
      SLD   3;	// shift left 3 bits to achieve pointer format
      LAR1;	// load adressregister 1 with pointer
      L     DBD [AR1,P#0.0];	// load position from DataBlock
      T     #tmp_di_ChkPosValHo;	// Transfer to temp for window check
      L     DBD [AR1,P#4.0];
      +D;
      T     #tmp_di_ChkPosValHu;
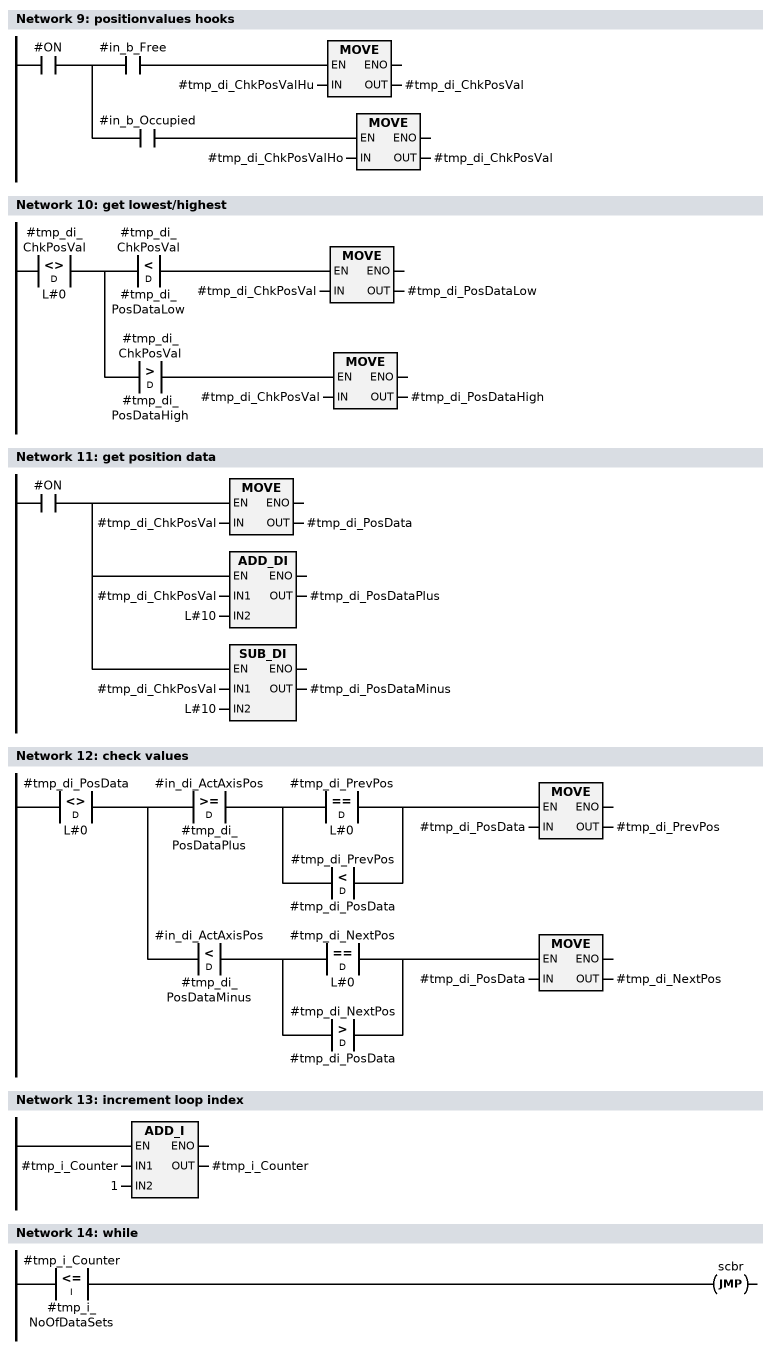
NETWORK
TITLE = positionvalues hooks
      A     #ON;
      =     L 65.0;
      A     L 65.0;
      A     #in_b_Free;
      JNB   _014;
      L     #tmp_di_ChkPosValHu;
      T     #tmp_di_ChkPosVal;
_014: NOP   0;
      A     L 65.0;
      A     #in_b_Occupied;
      JNB   _015;
      L     #tmp_di_ChkPosValHo;
      T     #tmp_di_ChkPosVal;
_015: NOP   0;
NETWORK
TITLE = get lowest/highest
      L     #tmp_di_ChkPosVal;
      L     L#0;
      <>D;
      =     L 65.0;
      A     L 65.0;
      A(;
      L     #tmp_di_ChkPosVal;
      L     #tmp_di_PosDataLow;
      <D;
      );
      JNB   _016;
      L     #tmp_di_ChkPosVal;
      T     #tmp_di_PosDataLow;
_016: NOP   0;
      A     L 65.0;
      A(;
      L     #tmp_di_ChkPosVal;
      L     #tmp_di_PosDataHigh;
      >D;
      );
      JNB   _017;
      L     #tmp_di_ChkPosVal;
      T     #tmp_di_PosDataHigh;
_017: NOP   0;
NETWORK
TITLE = get position data
      A     #ON;
      =     L 65.0;
      A     L 65.0;
      JNB   _018;
      L     #tmp_di_ChkPosVal;
      T     #tmp_di_PosData;
_018: NOP   0;
      A     L 65.0;
      JNB   _019;
      L     #tmp_di_ChkPosVal;
      L     L#10;
      +D;
      T     #tmp_di_PosDataPlus;
_019: NOP   0;
      A     L 65.0;
      JNB   _01a;
      L     #tmp_di_ChkPosVal;
      L     L#10;
      -D;
      T     #tmp_di_PosDataMinus;
_01a: NOP   0;
NETWORK
TITLE = check values
      L     #tmp_di_PosData;
      L     L#0;
      <>D;
      =     L 65.0;
      A     L 65.0;
      A(;
      L     #in_di_ActAxisPos;
      L     #tmp_di_PosDataPlus;
      >=D;
      );
      A(;
      O(;
      L     #tmp_di_PrevPos;
      L     L#0;
      ==D;
      );
      O(;
      L     #tmp_di_PrevPos;
      L     #tmp_di_PosData;
      <D;
      );
      );
      JNB   _01b;
      L     #tmp_di_PosData;
      T     #tmp_di_PrevPos;
_01b: NOP   0;
      A     L 65.0;
      A(;
      L     #in_di_ActAxisPos;
      L     #tmp_di_PosDataMinus;
      <D;
      );
      A(;
      O(;
      L     #tmp_di_NextPos;
      L     L#0;
      ==D;
      );
      O(;
      L     #tmp_di_NextPos;
      L     #tmp_di_PosData;
      >D;
      );
      );
      JNB   _01c;
      L     #tmp_di_PosData;
      T     #tmp_di_NextPos;
_01c: NOP   0;
NETWORK
TITLE = increment loop index
      L     #tmp_i_Counter;
      L     1;
      +I;
      T     #tmp_i_Counter;
      NOP   0;
NETWORK
TITLE = while 
      L     #tmp_i_Counter;
      L     #tmp_i_NoOfDataSets;
      <=I;
      JC    scbr;
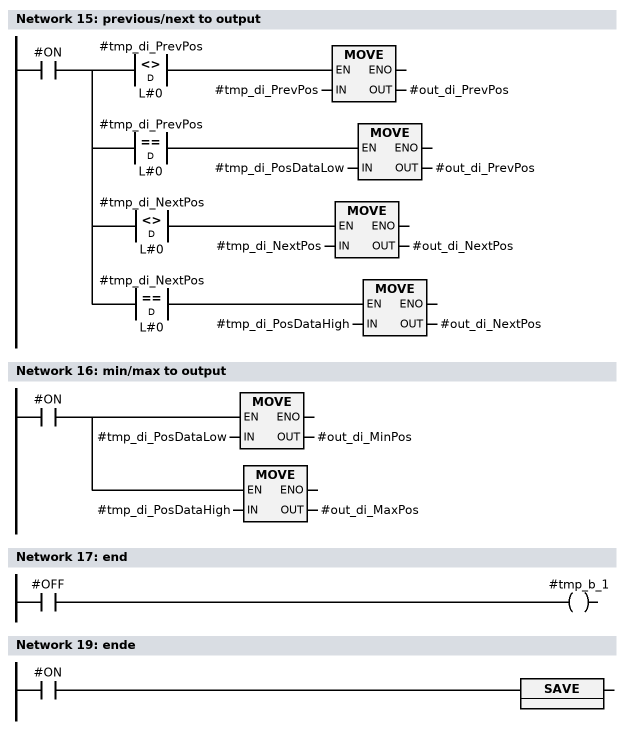
NETWORK
TITLE = previous/next to output
      A     #ON;
      =     L 65.0;
      A     L 65.0;
      A(;
      L     #tmp_di_PrevPos;
      L     L#0;
      <>D;
      );
      JNB   _01d;
      L     #tmp_di_PrevPos;
      T     #out_di_PrevPos;
_01d: NOP   0;
      A     L 65.0;
      A(;
      L     #tmp_di_PrevPos;
      L     L#0;
      ==D;
      );
      JNB   _01e;
      L     #tmp_di_PosDataLow;
      T     #out_di_PrevPos;
_01e: NOP   0;
      A     L 65.0;
      A(;
      L     #tmp_di_NextPos;
      L     L#0;
      <>D;
      );
      JNB   _01f;
      L     #tmp_di_NextPos;
      T     #out_di_NextPos;
_01f: NOP   0;
      A     L 65.0;
      A(;
      L     #tmp_di_NextPos;
      L     L#0;
      ==D;
      );
      JNB   _020;
      L     #tmp_di_PosDataHigh;
      T     #out_di_NextPos;
_020: NOP   0;
NETWORK
TITLE = min/max to output
      A     #ON;
      =     L 65.0;
      A     L 65.0;
      JNB   _021;
      L     #tmp_di_PosDataLow;
      T     #out_di_MinPos;
_021: NOP   0;
      A     L 65.0;
      JNB   _022;
      L     #tmp_di_PosDataHigh;
      T     #out_di_MaxPos;
_022: NOP   0;
NETWORK
TITLE = end
ende: A     #OFF;
      =     #tmp_b_1;
NETWORK
TITLE = restore register
      LAR1  #Save_AR1;
      LAR2  #Save_AR2;
NETWORK
TITLE = ende
      A     #ON;
      SAVE;
END_FUNCTION

FUNCTION "Scan_TEL" : VOID	// FC 27
TITLE = scan positions teleskops
VERSION : 1.1
VAR_INPUT
  in_di_ValCenter : DINT ;
  in_di_ValPos1 : DINT ;
  in_di_ValPos2 : DINT ;
  in_di_ValPos3 : DINT ;
  in_di_ActaPosVal : DINT ;
  in_AreaWin : DINT ;
  in_PosWin : DINT ;
END_VAR
VAR_OUTPUT
  out_i_AreaNo : INT ;
  out_b_InArea : BOOL ;
  out_b_InPos : BOOL ;
END_VAR
VAR_TEMP
  tmp_di_AbsDiff : DINT ;
  tmp_di_ChkWin : DINT ;
  ON : BOOL ;
  tmp_b_AreaCenter : BOOL ;
  tmp_b_PosCenter : BOOL ;
  tmp_b_AreaPos1 : BOOL ;
  tmp_b_PosPos1 : BOOL ;
  tmp_b_AreaPos2 : BOOL ;
  tmp_b_PosPos2 : BOOL ;
  tmp_b_AreaPos3 : BOOL ;
  tmp_b_PosPos3 : BOOL ;
  tmp_b_Rear : BOOL ;
  tmp_b_Front : BOOL ;
END_VAR
BEGIN
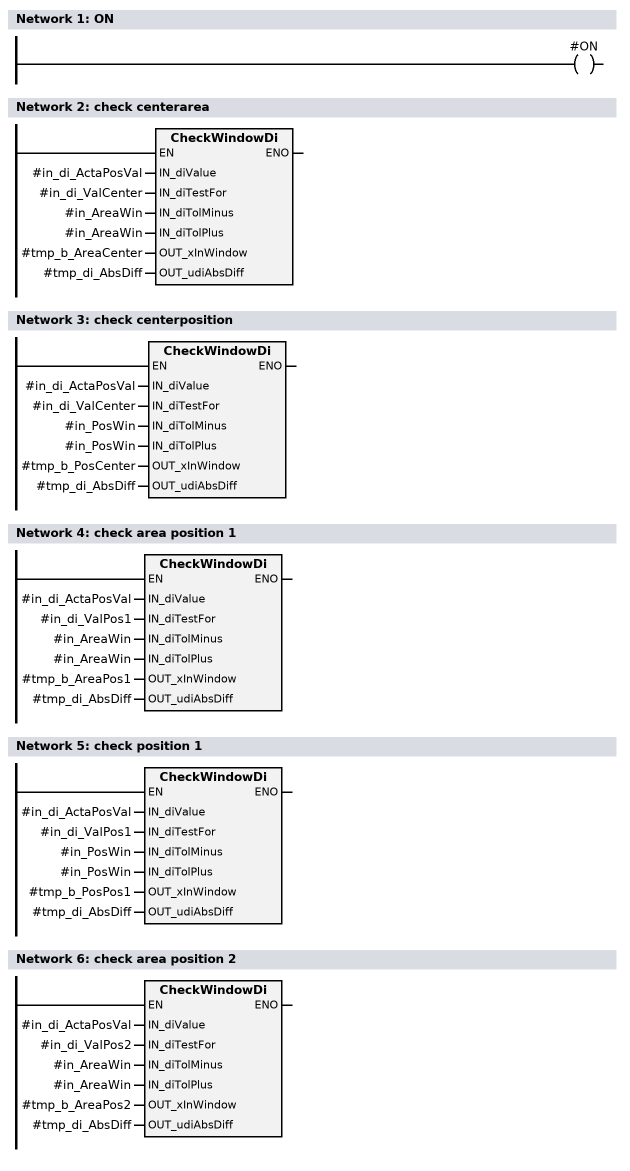
NETWORK
TITLE = ON
      SET;
      =     #ON;
NETWORK
TITLE = check centerarea
      CALL  "CheckWindowDi" (
           IN_diValue               := #in_di_ActaPosVal,
           IN_diTestFor             := #in_di_ValCenter,
           IN_diTolMinus            := #in_AreaWin,
           IN_diTolPlus             := #in_AreaWin,
           OUT_xInWindow            := #tmp_b_AreaCenter,
           OUT_udiAbsDiff           := #tmp_di_AbsDiff);
      NOP   0;
NETWORK
TITLE = check centerposition
      CALL  "CheckWindowDi" (
           IN_diValue               := #in_di_ActaPosVal,
           IN_diTestFor             := #in_di_ValCenter,
           IN_diTolMinus            := #in_PosWin,
           IN_diTolPlus             := #in_PosWin,
           OUT_xInWindow            := #tmp_b_PosCenter,
           OUT_udiAbsDiff           := #tmp_di_AbsDiff);
      NOP   0;
NETWORK
TITLE = check area position 1 
      CALL  "CheckWindowDi" (
           IN_diValue               := #in_di_ActaPosVal,
           IN_diTestFor             := #in_di_ValPos1,
           IN_diTolMinus            := #in_AreaWin,
           IN_diTolPlus             := #in_AreaWin,
           OUT_xInWindow            := #tmp_b_AreaPos1,
           OUT_udiAbsDiff           := #tmp_di_AbsDiff);
      NOP   0;
NETWORK
TITLE = check position 1
      CALL  "CheckWindowDi" (
           IN_diValue               := #in_di_ActaPosVal,
           IN_diTestFor             := #in_di_ValPos1,
           IN_diTolMinus            := #in_PosWin,
           IN_diTolPlus             := #in_PosWin,
           OUT_xInWindow            := #tmp_b_PosPos1,
           OUT_udiAbsDiff           := #tmp_di_AbsDiff);
      NOP   0;
NETWORK
TITLE = check area position 2 
      CALL  "CheckWindowDi" (
           IN_diValue               := #in_di_ActaPosVal,
           IN_diTestFor             := #in_di_ValPos2,
           IN_diTolMinus            := #in_AreaWin,
           IN_diTolPlus             := #in_AreaWin,
           OUT_xInWindow            := #tmp_b_AreaPos2,
           OUT_udiAbsDiff           := #tmp_di_AbsDiff);
      NOP   0;
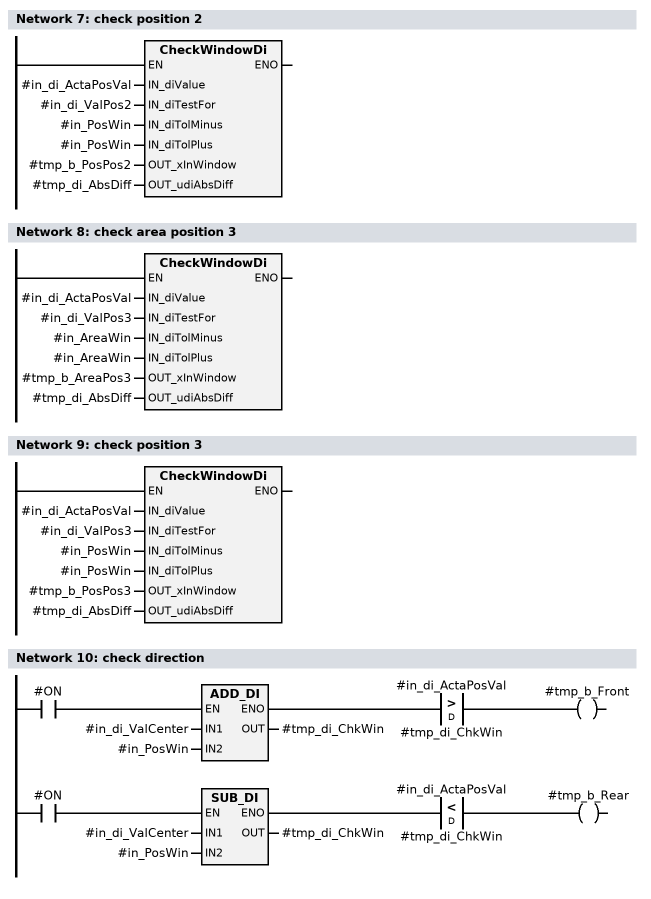
NETWORK
TITLE = check position 2
      CALL  "CheckWindowDi" (
           IN_diValue               := #in_di_ActaPosVal,
           IN_diTestFor             := #in_di_ValPos2,
           IN_diTolMinus            := #in_PosWin,
           IN_diTolPlus             := #in_PosWin,
           OUT_xInWindow            := #tmp_b_PosPos2,
           OUT_udiAbsDiff           := #tmp_di_AbsDiff);
      NOP   0;
NETWORK
TITLE = check area position 3 
      CALL  "CheckWindowDi" (
           IN_diValue               := #in_di_ActaPosVal,
           IN_diTestFor             := #in_di_ValPos3,
           IN_diTolMinus            := #in_AreaWin,
           IN_diTolPlus             := #in_AreaWin,
           OUT_xInWindow            := #tmp_b_AreaPos3,
           OUT_udiAbsDiff           := #tmp_di_AbsDiff);
      NOP   0;
NETWORK
TITLE = check position 3
      CALL  "CheckWindowDi" (
           IN_diValue               := #in_di_ActaPosVal,
           IN_diTestFor             := #in_di_ValPos3,
           IN_diTolMinus            := #in_PosWin,
           IN_diTolPlus             := #in_PosWin,
           OUT_xInWindow            := #tmp_b_PosPos3,
           OUT_udiAbsDiff           := #tmp_di_AbsDiff);
      NOP   0;
NETWORK
TITLE = check direction
      A     #ON;
      =     L 10.0;
      A(;
      A     L 10.0;
      JNB   _001;
      L     #in_di_ValCenter;
      L     #in_PosWin;
      +D;
      T     #tmp_di_ChkWin;
      AN    OV;
      SAVE;
      CLR;
_001: A     BR;
      );
      A(;
      L     #in_di_ActaPosVal;
      L     #tmp_di_ChkWin;
      >D;
      );
      =     #tmp_b_Front;
      A(;
      A     L 10.0;
      JNB   _002;
      L     #in_di_ValCenter;
      L     #in_PosWin;
      -D;
      T     #tmp_di_ChkWin;
      AN    OV;
      SAVE;
      CLR;
_002: A     BR;
      );
      A(;
      L     #in_di_ActaPosVal;
      L     #tmp_di_ChkWin;
      <D;
      );
      =     #tmp_b_Rear;
